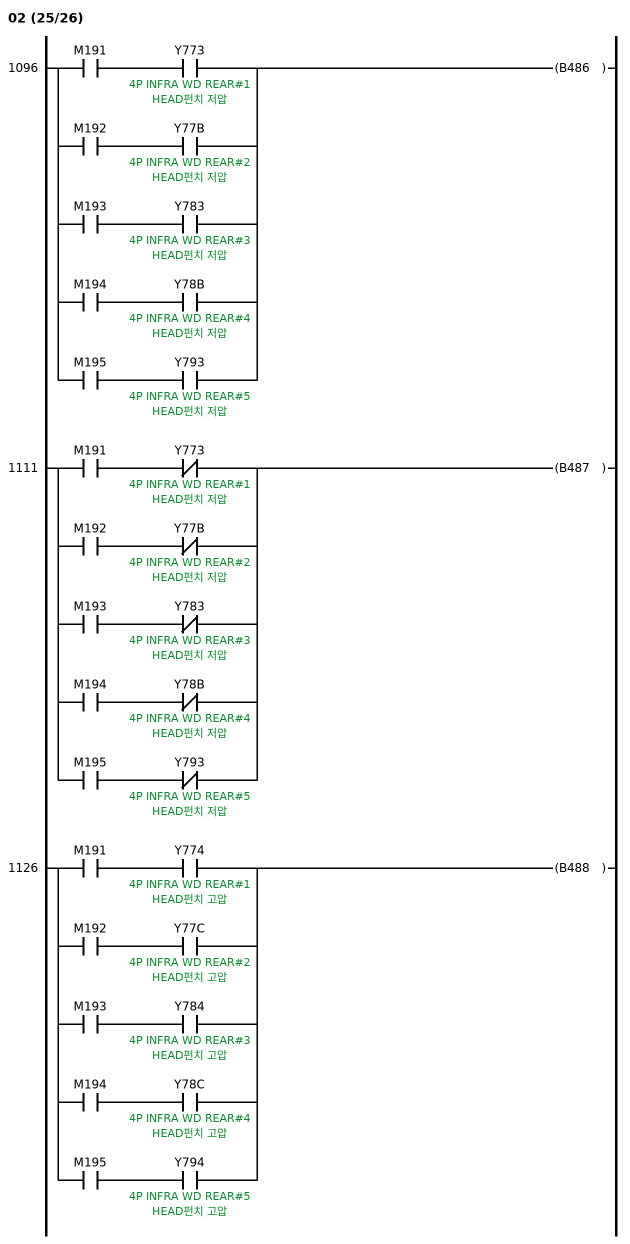
1096  LD      M191
      AND     Y773  ; 4P INFRA WD REAR#1 HEAD펀치 저압
      LD      M192
      AND     Y77B  ; 4P INFRA WD REAR#2 HEAD펀치 저압
      ORB
      LD      M193
      AND     Y783  ; 4P INFRA WD REAR#3 HEAD펀치 저압
      ORB
      LD      M194
      AND     Y78B  ; 4P INFRA WD REAR#4 HEAD펀치 저압
      ORB
      LD      M195
      AND     Y793  ; 4P INFRA WD REAR#5 HEAD펀치 저압
      ORB
      OUT     B486
1111  LD      M191
      ANI     Y773  ; 4P INFRA WD REAR#1 HEAD펀치 저압
      LD      M192
      ANI     Y77B  ; 4P INFRA WD REAR#2 HEAD펀치 저압
      ORB
      LD      M193
      ANI     Y783  ; 4P INFRA WD REAR#3 HEAD펀치 저압
      ORB
      LD      M194
      ANI     Y78B  ; 4P INFRA WD REAR#4 HEAD펀치 저압
      ORB
      LD      M195
      ANI     Y793  ; 4P INFRA WD REAR#5 HEAD펀치 저압
      ORB
      OUT     B487
1126  LD      M191
      AND     Y774  ; 4P INFRA WD REAR#1 HEAD펀치 고압
      LD      M192
      AND     Y77C  ; 4P INFRA WD REAR#2 HEAD펀치 고압
      ORB
      LD      M193
      AND     Y784  ; 4P INFRA WD REAR#3 HEAD펀치 고압
      ORB
      LD      M194
      AND     Y78C  ; 4P INFRA WD REAR#4 HEAD펀치 고압
      ORB
      LD      M195
      AND     Y794  ; 4P INFRA WD REAR#5 HEAD펀치 고압
      ORB
      OUT     B488
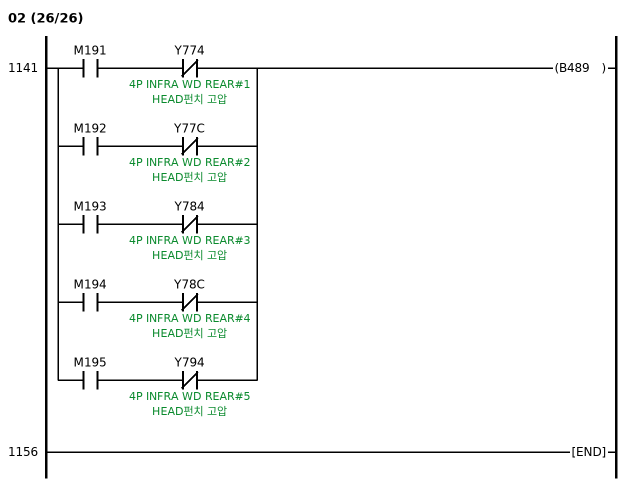
1141  LD      M191
      ANI     Y774  ; 4P INFRA WD REAR#1 HEAD펀치 고압
      LD      M192
      ANI     Y77C  ; 4P INFRA WD REAR#2 HEAD펀치 고압
      ORB
      LD      M193
      ANI     Y784  ; 4P INFRA WD REAR#3 HEAD펀치 고압
      ORB
      LD      M194
      ANI     Y78C  ; 4P INFRA WD REAR#4 HEAD펀치 고압
      ORB
      LD      M195
      ANI     Y794  ; 4P INFRA WD REAR#5 HEAD펀치 고압
      ORB
      OUT     B489
1156  END
END_PROGRAM

PROGRAM 03  // OUTPUT
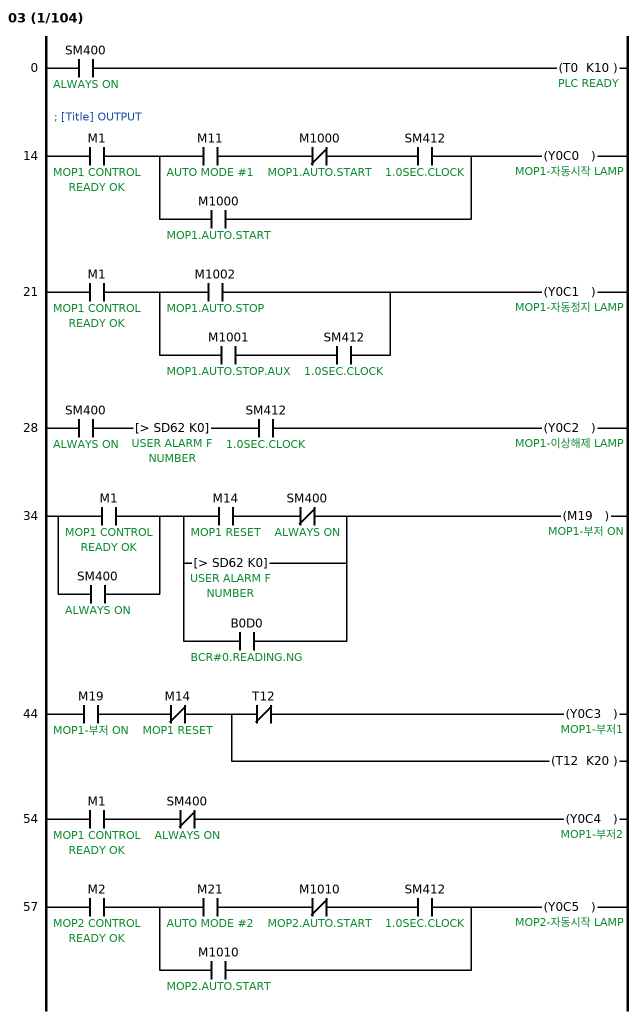
0     LD      SM400  ; ALWAYS ON
      OUT     T0 K10  ; PLC READY
; [Title] OUTPUT
14    LD      M1  ; MOP1 CONTROL READY OK
      LD      M11  ; AUTO MODE #1
      ANI     M1000  ; MOP1.AUTO.START
      AND     SM412  ; 1.0SEC.CLOCK
      OR      M1000  ; MOP1.AUTO.START
      ANB
      OUT     Y0C0  ; MOP1-자동시작 LAMP
21    LD      M1  ; MOP1 CONTROL READY OK
      LD      M1002  ; MOP1.AUTO.STOP
      LD      M1001  ; MOP1.AUTO.STOP.AUX
      AND     SM412  ; 1.0SEC.CLOCK
      ORB
      ANB
      OUT     Y0C1  ; MOP1-자동정지 LAMP
28    LD      SM400  ; ALWAYS ON
      AND>    SD62 K0  ; USER ALARM F NUMBER
      AND     SM412  ; 1.0SEC.CLOCK
      OUT     Y0C2  ; MOP1-이상해제 LAMP
34    LD      M1  ; MOP1 CONTROL READY OK
      OR      SM400  ; ALWAYS ON
      LD      M14  ; MOP1 RESET
      ANI     SM400  ; ALWAYS ON
      OR>     SD62 K0  ; USER ALARM F NUMBER
      OR      B0D0  ; BCR#0.READING.NG
      ANB
      OUT     M19  ; MOP1-부저 ON
44    LD      M19  ; MOP1-부저 ON
      ANI     M14  ; MOP1 RESET
      MPS
      ANI     T12
      OUT     Y0C3  ; MOP1-부저1
      MPP
      OUT     T12 K20
54    LD      M1  ; MOP1 CONTROL READY OK
      ANI     SM400  ; ALWAYS ON
      OUT     Y0C4  ; MOP1-부저2
57    LD      M2  ; MOP2 CONTROL READY OK
      LD      M21  ; AUTO MODE #2
      ANI     M1010  ; MOP2.AUTO.START
      AND     SM412  ; 1.0SEC.CLOCK
      OR      M1010  ; MOP2.AUTO.START
      ANB
      OUT     Y0C5  ; MOP2-자동시작 LAMP
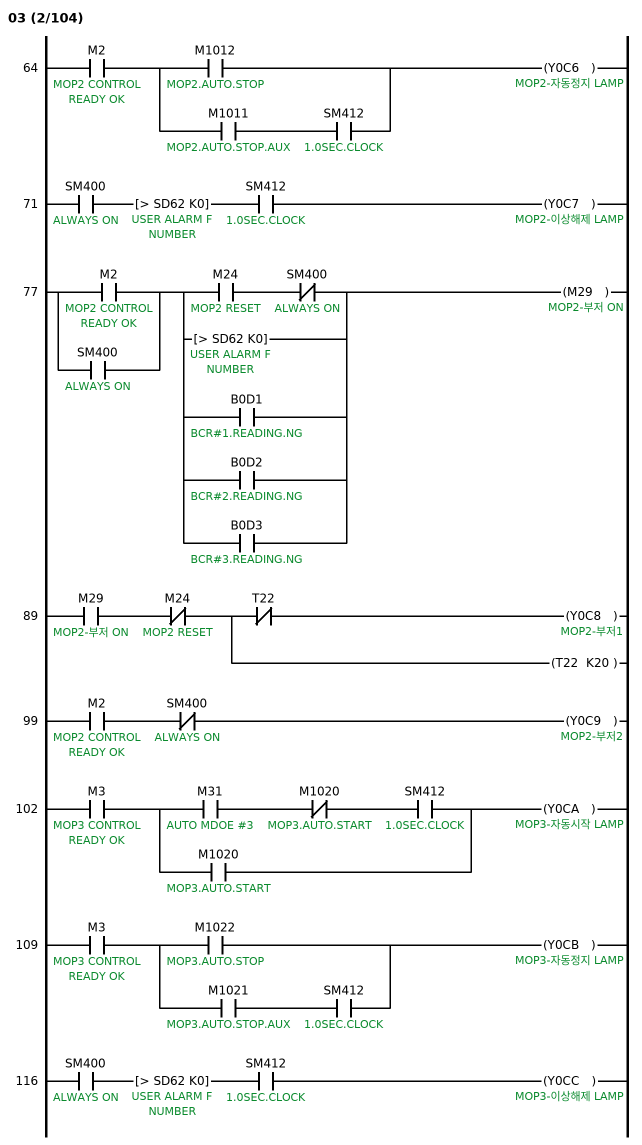
64    LD      M2  ; MOP2 CONTROL READY OK
      LD      M1012  ; MOP2.AUTO.STOP
      LD      M1011  ; MOP2.AUTO.STOP.AUX
      AND     SM412  ; 1.0SEC.CLOCK
      ORB
      ANB
      OUT     Y0C6  ; MOP2-자동정지 LAMP
71    LD      SM400  ; ALWAYS ON
      AND>    SD62 K0  ; USER ALARM F NUMBER
      AND     SM412  ; 1.0SEC.CLOCK
      OUT     Y0C7  ; MOP2-이상해제 LAMP
77    LD      M2  ; MOP2 CONTROL READY OK
      OR      SM400  ; ALWAYS ON
      LD      M24  ; MOP2 RESET
      ANI     SM400  ; ALWAYS ON
      OR>     SD62 K0  ; USER ALARM F NUMBER
      OR      B0D1  ; BCR#1.READING.NG
      OR      B0D2  ; BCR#2.READING.NG
      OR      B0D3  ; BCR#3.READING.NG
      ANB
      OUT     M29  ; MOP2-부저 ON
89    LD      M29  ; MOP2-부저 ON
      ANI     M24  ; MOP2 RESET
      MPS
      ANI     T22
      OUT     Y0C8  ; MOP2-부저1
      MPP
      OUT     T22 K20
99    LD      M2  ; MOP2 CONTROL READY OK
      ANI     SM400  ; ALWAYS ON
      OUT     Y0C9  ; MOP2-부저2
102   LD      M3  ; MOP3 CONTROL READY OK
      LD      M31  ; AUTO MDOE #3
      ANI     M1020  ; MOP3.AUTO.START
      AND     SM412  ; 1.0SEC.CLOCK
      OR      M1020  ; MOP3.AUTO.START
      ANB
      OUT     Y0CA  ; MOP3-자동시작 LAMP
109   LD      M3  ; MOP3 CONTROL READY OK
      LD      M1022  ; MOP3.AUTO.STOP
      LD      M1021  ; MOP3.AUTO.STOP.AUX
      AND     SM412  ; 1.0SEC.CLOCK
      ORB
      ANB
      OUT     Y0CB  ; MOP3-자동정지 LAMP
116   LD      SM400  ; ALWAYS ON
      AND>    SD62 K0  ; USER ALARM F NUMBER
      AND     SM412  ; 1.0SEC.CLOCK
      OUT     Y0CC  ; MOP3-이상해제 LAMP
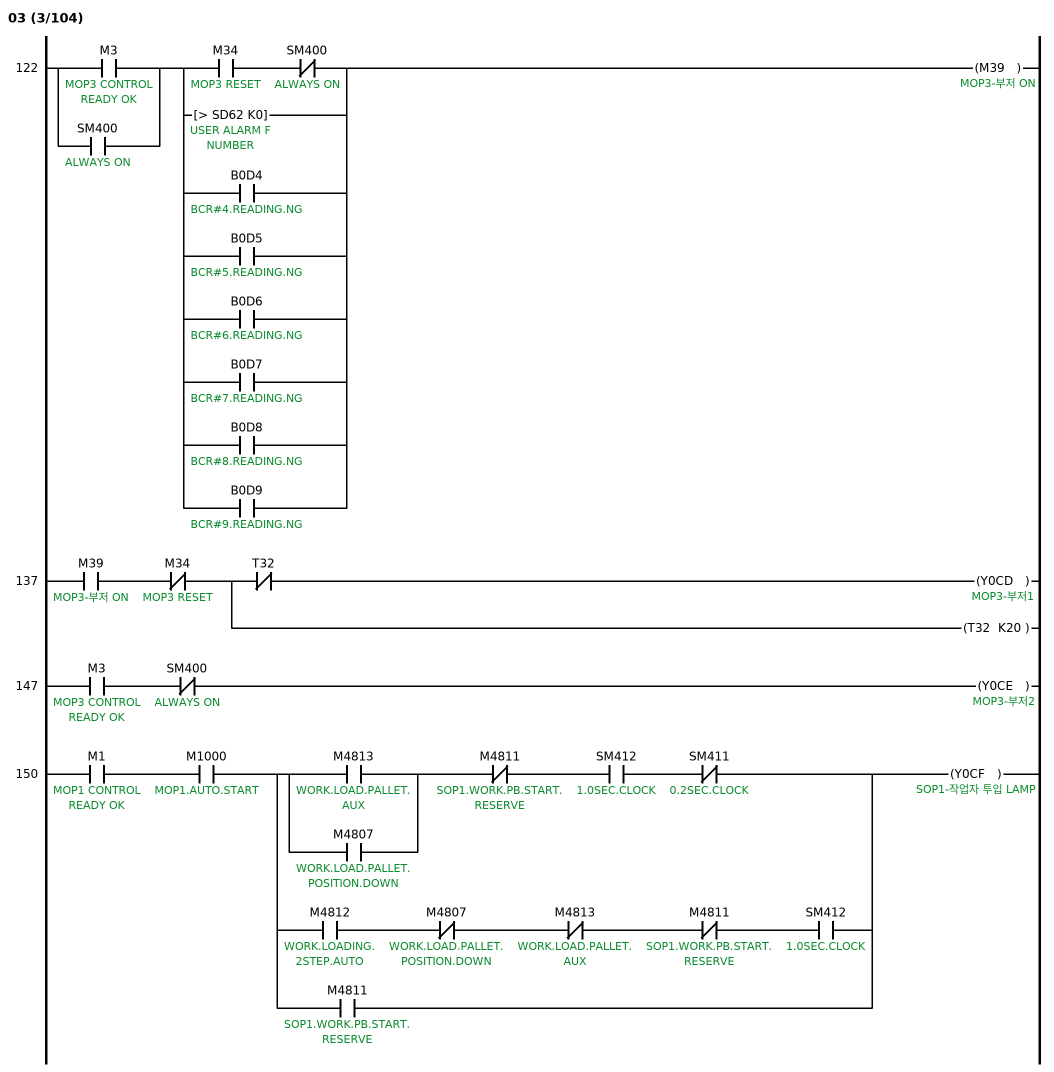
122   LD      M3  ; MOP3 CONTROL READY OK
      OR      SM400  ; ALWAYS ON
      LD      M34  ; MOP3 RESET
      ANI     SM400  ; ALWAYS ON
      OR>     SD62 K0  ; USER ALARM F NUMBER
      OR      B0D4  ; BCR#4.READING.NG
      OR      B0D5  ; BCR#5.READING.NG
      OR      B0D6  ; BCR#6.READING.NG
      OR      B0D7  ; BCR#7.READING.NG
      OR      B0D8  ; BCR#8.READING.NG
      OR      B0D9  ; BCR#9.READING.NG
      ANB
      OUT     M39  ; MOP3-부저 ON
137   LD      M39  ; MOP3-부저 ON
      ANI     M34  ; MOP3 RESET
      MPS
      ANI     T32
      OUT     Y0CD  ; MOP3-부저1
      MPP
      OUT     T32 K20
147   LD      M3  ; MOP3 CONTROL READY OK
      ANI     SM400  ; ALWAYS ON
      OUT     Y0CE  ; MOP3-부저2
150   LD      M1  ; MOP1 CONTROL READY OK
      AND     M1000  ; MOP1.AUTO.START
      LD      M4813  ; WORK.LOAD.PALLET.AUX
      OR      M4807  ; WORK.LOAD.PALLET.POSITION.DOWN
      ANI     M4811  ; SOP1.WORK.PB.START.RESERVE
      AND     SM412  ; 1.0SEC.CLOCK
      ANI     SM411  ; 0.2SEC.CLOCK
      LD      M4812  ; WORK.LOADING.2STEP.AUTO
      ANI     M4807  ; WORK.LOAD.PALLET.POSITION.DOWN
      ANI     M4813  ; WORK.LOAD.PALLET.AUX
      ANI     M4811  ; SOP1.WORK.PB.START.RESERVE
      AND     SM412  ; 1.0SEC.CLOCK
      ORB
      OR      M4811  ; SOP1.WORK.PB.START.RESERVE
      ANB
      OUT     Y0CF  ; SOP1-작업자 투입 LAMP
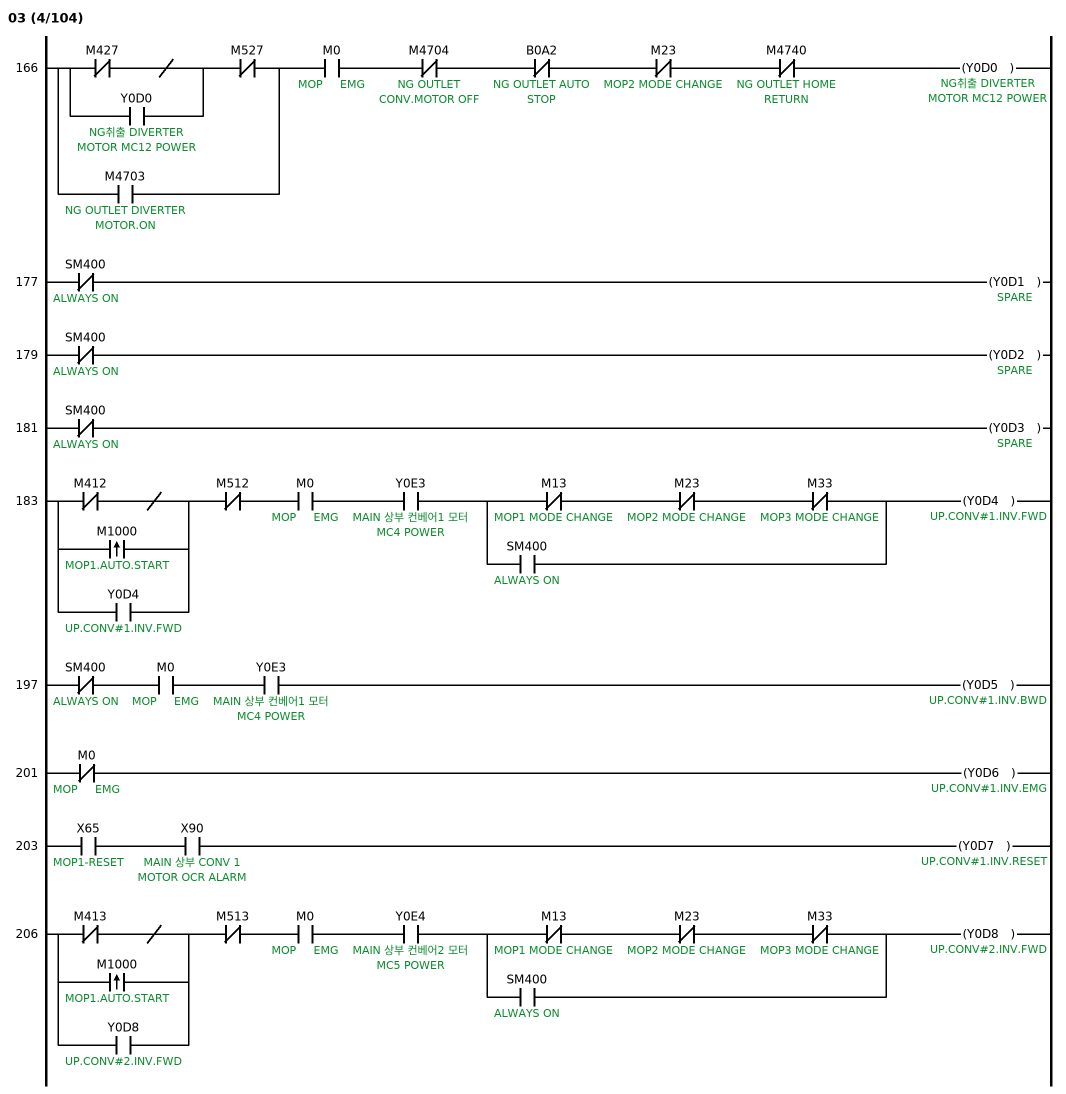
166   LDI     M427
      INV
      OR      Y0D0  ; NG취출 DIVERTER MOTOR MC12 POWER
      ANI     M527
      OR      M4703  ; NG OUTLET DIVERTER MOTOR.ON
      AND     M0  ; MOP     EMG
      ANI     M4704  ; NG OUTLET CONV.MOTOR OFF
      ANI     B0A2  ; NG OUTLET AUTO STOP
      ANI     M23  ; MOP2 MODE CHANGE
      ANI     M4740  ; NG OUTLET HOME RETURN
      OUT     Y0D0  ; NG취출 DIVERTER MOTOR MC12 POWER
177   LDI     SM400  ; ALWAYS ON
      OUT     Y0D1  ; SPARE
179   LDI     SM400  ; ALWAYS ON
      OUT     Y0D2  ; SPARE
181   LDI     SM400  ; ALWAYS ON
      OUT     Y0D3  ; SPARE
183   LDI     M412
      INV
      ORP     M1000  ; MOP1.AUTO.START
      OR      Y0D4  ; UP.CONV#1.INV.FWD
      ANI     M512
      AND     M0  ; MOP     EMG
      AND     Y0E3  ; MAIN 상부 컨베어1 모터 MC4 POWER
      LDI     M13  ; MOP1 MODE CHANGE
      ANI     M23  ; MOP2 MODE CHANGE
      ANI     M33  ; MOP3 MODE CHANGE
      OR      SM400  ; ALWAYS ON
      ANB
      OUT     Y0D4  ; UP.CONV#1.INV.FWD
197   LDI     SM400  ; ALWAYS ON
      AND     M0  ; MOP     EMG
      AND     Y0E3  ; MAIN 상부 컨베어1 모터 MC4 POWER
      OUT     Y0D5  ; UP.CONV#1.INV.BWD
201   LDI     M0  ; MOP     EMG
      OUT     Y0D6  ; UP.CONV#1.INV.EMG
203   LD      X65  ; MOP1-RESET
      AND     X90  ; MAIN 상부 CONV 1 MOTOR OCR ALARM
      OUT     Y0D7  ; UP.CONV#1.INV.RESET
206   LDI     M413
      INV
      ORP     M1000  ; MOP1.AUTO.START
      OR      Y0D8  ; UP.CONV#2.INV.FWD
      ANI     M513
      AND     M0  ; MOP     EMG
      AND     Y0E4  ; MAIN 상부 컨베어2 모터 MC5 POWER
      LDI     M13  ; MOP1 MODE CHANGE
      ANI     M23  ; MOP2 MODE CHANGE
      ANI     M33  ; MOP3 MODE CHANGE
      OR      SM400  ; ALWAYS ON
      ANB
      OUT     Y0D8  ; UP.CONV#2.INV.FWD
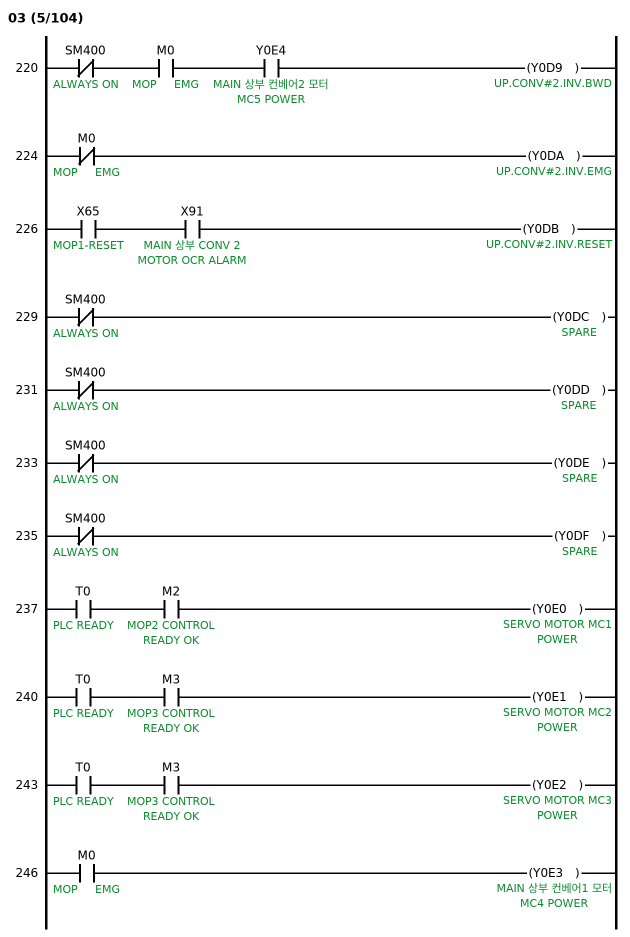
220   LDI     SM400  ; ALWAYS ON
      AND     M0  ; MOP     EMG
      AND     Y0E4  ; MAIN 상부 컨베어2 모터 MC5 POWER
      OUT     Y0D9  ; UP.CONV#2.INV.BWD
224   LDI     M0  ; MOP     EMG
      OUT     Y0DA  ; UP.CONV#2.INV.EMG
226   LD      X65  ; MOP1-RESET
      AND     X91  ; MAIN 상부 CONV 2 MOTOR OCR ALARM
      OUT     Y0DB  ; UP.CONV#2.INV.RESET
229   LDI     SM400  ; ALWAYS ON
      OUT     Y0DC  ; SPARE
231   LDI     SM400  ; ALWAYS ON
      OUT     Y0DD  ; SPARE
233   LDI     SM400  ; ALWAYS ON
      OUT     Y0DE  ; SPARE
235   LDI     SM400  ; ALWAYS ON
      OUT     Y0DF  ; SPARE
237   LD      T0  ; PLC READY
      AND     M2  ; MOP2 CONTROL READY OK
      OUT     Y0E0  ; SERVO MOTOR MC1 POWER
240   LD      T0  ; PLC READY
      AND     M3  ; MOP3 CONTROL READY OK
      OUT     Y0E1  ; SERVO MOTOR MC2 POWER
243   LD      T0  ; PLC READY
      AND     M3  ; MOP3 CONTROL READY OK
      OUT     Y0E2  ; SERVO MOTOR MC3 POWER
246   LD      M0  ; MOP     EMG
      OUT     Y0E3  ; MAIN 상부 컨베어1 모터 MC4 POWER
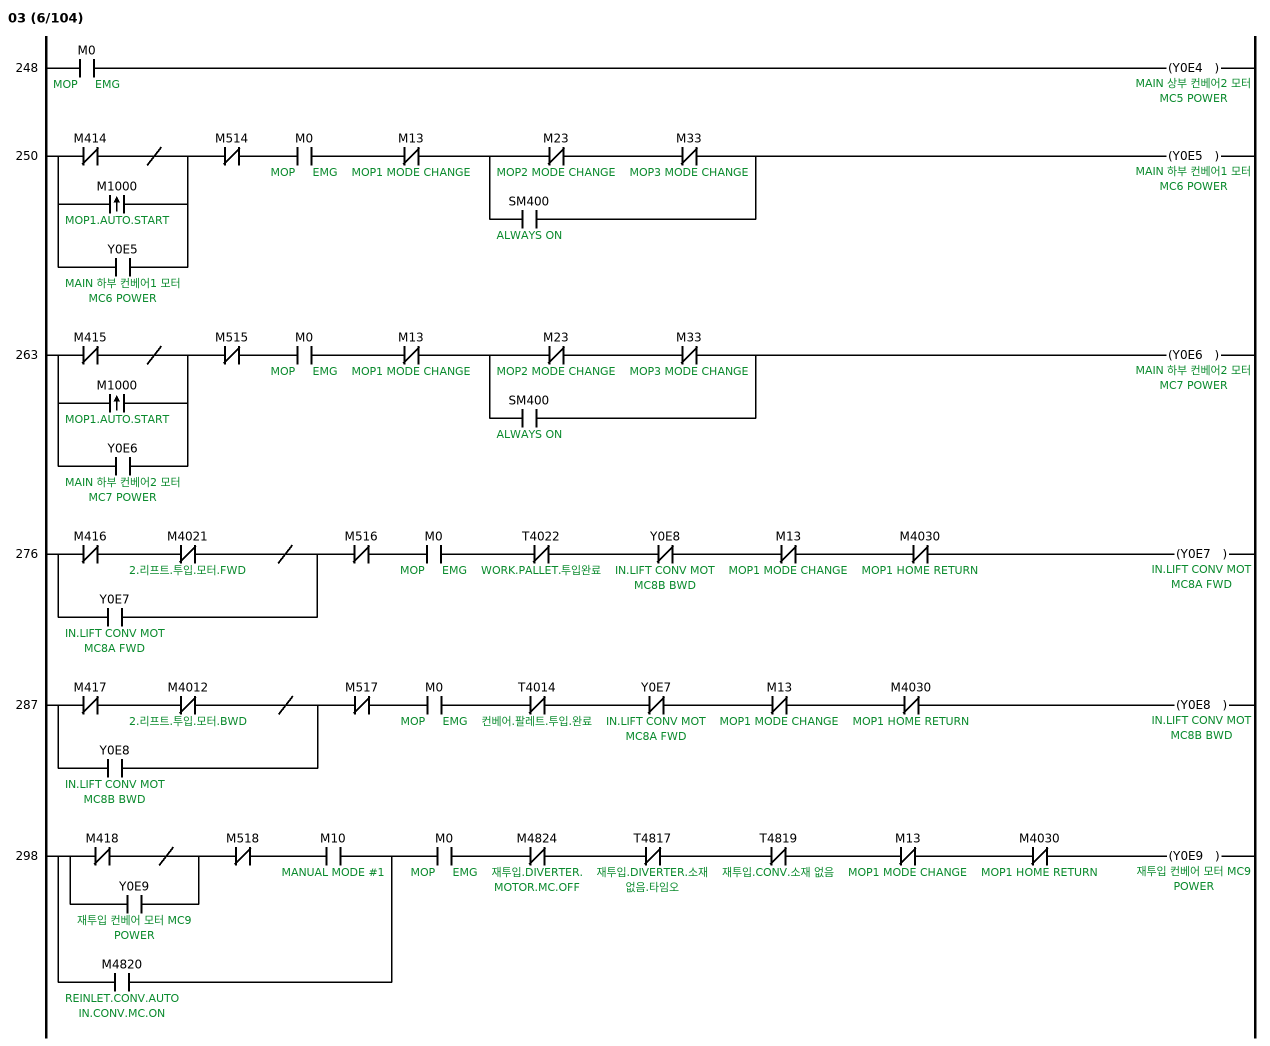
248   LD      M0  ; MOP     EMG
      OUT     Y0E4  ; MAIN 상부 컨베어2 모터 MC5 POWER
250   LDI     M414
      INV
      ORP     M1000  ; MOP1.AUTO.START
      OR      Y0E5  ; MAIN 하부 컨베어1 모터 MC6 POWER
      ANI     M514
      AND     M0  ; MOP     EMG
      ANI     M13  ; MOP1 MODE CHANGE
      LDI     M23  ; MOP2 MODE CHANGE
      ANI     M33  ; MOP3 MODE CHANGE
      OR      SM400  ; ALWAYS ON
      ANB
      OUT     Y0E5  ; MAIN 하부 컨베어1 모터 MC6 POWER
263   LDI     M415
      INV
      ORP     M1000  ; MOP1.AUTO.START
      OR      Y0E6  ; MAIN 하부 컨베어2 모터 MC7 POWER
      ANI     M515
      AND     M0  ; MOP     EMG
      ANI     M13  ; MOP1 MODE CHANGE
      LDI     M23  ; MOP2 MODE CHANGE
      ANI     M33  ; MOP3 MODE CHANGE
      OR      SM400  ; ALWAYS ON
      ANB
      OUT     Y0E6  ; MAIN 하부 컨베어2 모터 MC7 POWER
276   LDI     M416
      ANI     M4021  ; 2.리프트.투입.모터.FWD
      INV
      OR      Y0E7  ; IN.LIFT CONV MOT MC8A FWD
      ANI     M516
      AND     M0  ; MOP     EMG
      ANI     T4022  ; WORK.PALLET.투입완료
      ANI     Y0E8  ; IN.LIFT CONV MOT MC8B BWD
      ANI     M13  ; MOP1 MODE CHANGE
      ANI     M4030  ; MOP1 HOME RETURN
      OUT     Y0E7  ; IN.LIFT CONV MOT MC8A FWD
287   LDI     M417
      ANI     M4012  ; 2.리프트.투입.모터.BWD
      INV
      OR      Y0E8  ; IN.LIFT CONV MOT MC8B BWD
      ANI     M517
      AND     M0  ; MOP     EMG
      ANI     T4014  ; 컨베어.팔레트.투입.완료
      ANI     Y0E7  ; IN.LIFT CONV MOT MC8A FWD
      ANI     M13  ; MOP1 MODE CHANGE
      ANI     M4030  ; MOP1 HOME RETURN
      OUT     Y0E8  ; IN.LIFT CONV MOT MC8B BWD
298   LDI     M418
      INV
      OR      Y0E9  ; 재투입 컨베어 모터 MC9 POWER
      ANI     M518
      AND     M10  ; MANUAL MODE #1
      OR      M4820  ; REINLET.CONV.AUTO IN.CONV.MC.ON
      AND     M0  ; MOP     EMG
      ANI     M4824  ; 재투입.DIVERTER.MOTOR.MC.OFF
      ANI     T4817  ; 재투입.DIVERTER.소재 없음.타임오
      ANI     T4819  ; 재투입.CONV.소재 없음
      ANI     M13  ; MOP1 MODE CHANGE
      ANI     M4030  ; MOP1 HOME RETURN
      OUT     Y0E9  ; 재투입 컨베어 모터 MC9 POWER
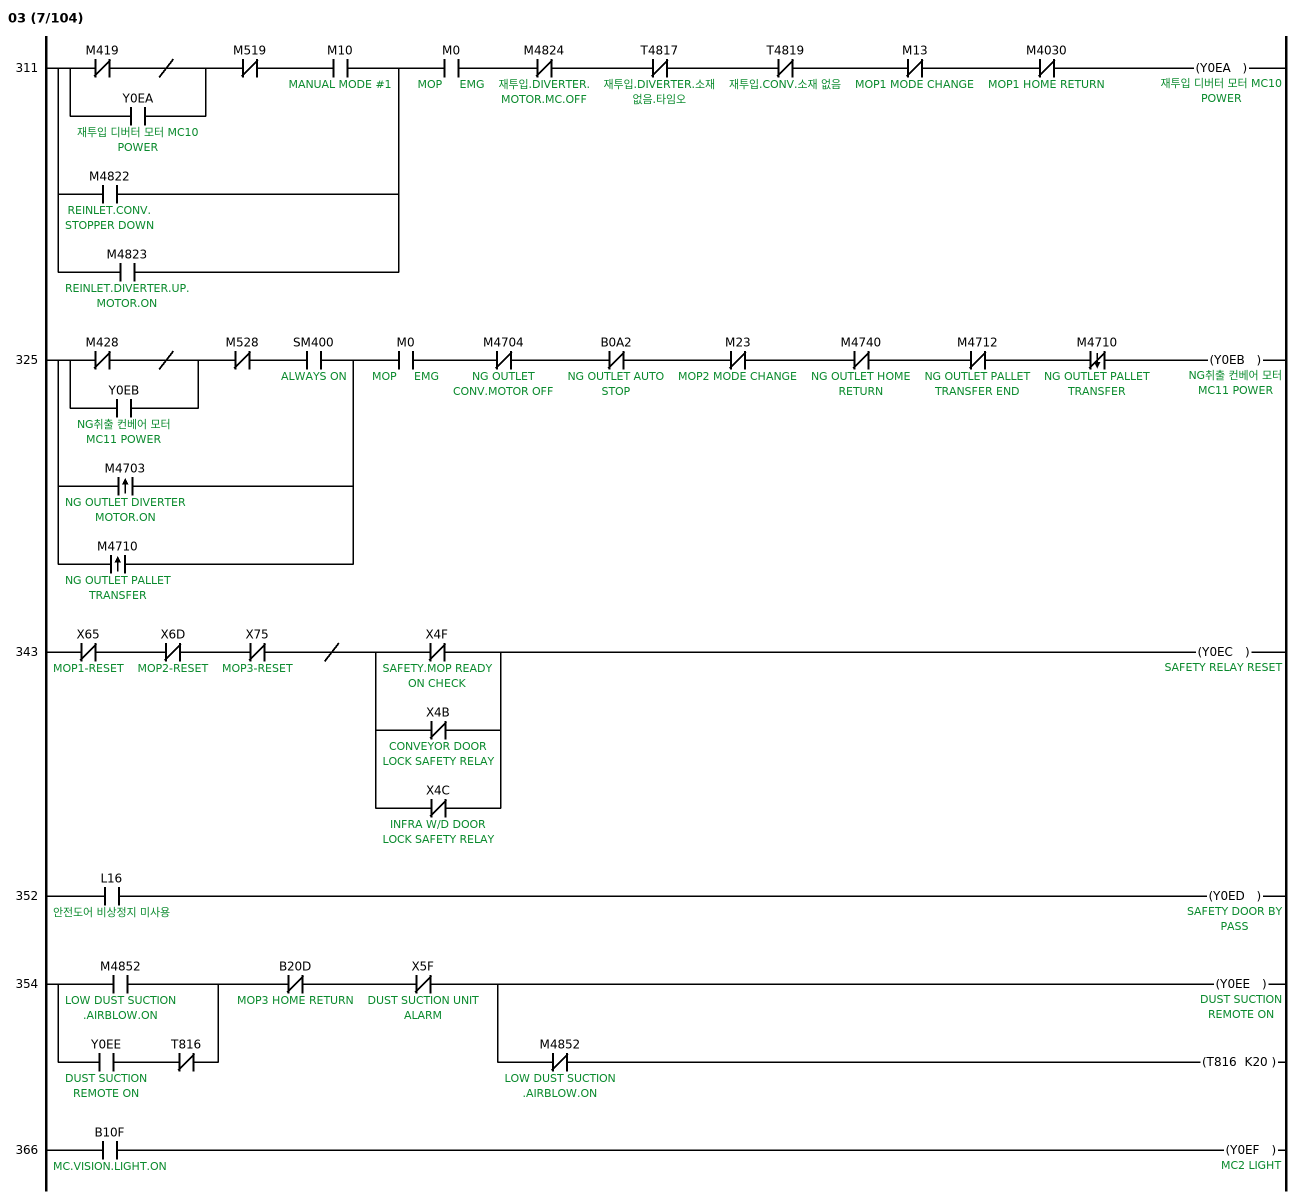
311   LDI     M419
      INV
      OR      Y0EA  ; 재투입 디버터 모터 MC10 POWER
      ANI     M519
      AND     M10  ; MANUAL MODE #1
      OR      M4822  ; REINLET.CONV.STOPPER DOWN
      OR      M4823  ; REINLET.DIVERTER.UP.MOTOR.ON
      AND     M0  ; MOP     EMG
      ANI     M4824  ; 재투입.DIVERTER.MOTOR.MC.OFF
      ANI     T4817  ; 재투입.DIVERTER.소재 없음.타임오
      ANI     T4819  ; 재투입.CONV.소재 없음
      ANI     M13  ; MOP1 MODE CHANGE
      ANI     M4030  ; MOP1 HOME RETURN
      OUT     Y0EA  ; 재투입 디버터 모터 MC10 POWER
325   LDI     M428
      INV
      OR      Y0EB  ; NG취출 컨베어 모터 MC11 POWER
      ANI     M528
      AND     SM400  ; ALWAYS ON
      ORP     M4703  ; NG OUTLET DIVERTER MOTOR.ON
      ORP     M4710  ; NG OUTLET PALLET TRANSFER
      AND     M0  ; MOP     EMG
      ANI     M4704  ; NG OUTLET CONV.MOTOR OFF
      ANI     B0A2  ; NG OUTLET AUTO STOP
      ANI     M23  ; MOP2 MODE CHANGE
      ANI     M4740  ; NG OUTLET HOME RETURN
      ANI     M4712  ; NG OUTLET PALLET TRANSFER END
      ANDFI   M4710  ; NG OUTLET PALLET TRANSFER
      OUT     Y0EB  ; NG취출 컨베어 모터 MC11 POWER
343   LDI     X65  ; MOP1-RESET
      ANI     X6D  ; MOP2-RESET
      ANI     X75  ; MOP3-RESET
      INV
      LDI     X4F  ; SAFETY.MOP READY ON CHECK
      ORI     X4B  ; CONVEYOR DOOR LOCK SAFETY RELAY
      ORI     X4C  ; INFRA W/D DOOR LOCK SAFETY RELAY
      ANB
      OUT     Y0EC  ; SAFETY RELAY RESET
352   LD      L16  ; 안전도어 비상정지 미사용
      OUT     Y0ED  ; SAFETY DOOR BY PASS
354   LD      M4852  ; LOW DUST SUCTION .AIRBLOW.ON
      LD      Y0EE  ; DUST SUCTION REMOTE ON
      ANI     T816
      ORB
      ANI     B20D  ; MOP3 HOME RETURN
      ANI     X5F  ; DUST SUCTION UNIT ALARM
      OUT     Y0EE  ; DUST SUCTION REMOTE ON
      ANI     M4852  ; LOW DUST SUCTION .AIRBLOW.ON
      OUT     T816 K20
366   LD      B10F  ; MC.VISION.LIGHT.ON
      OUT     Y0EF  ; MC2 LIGHT
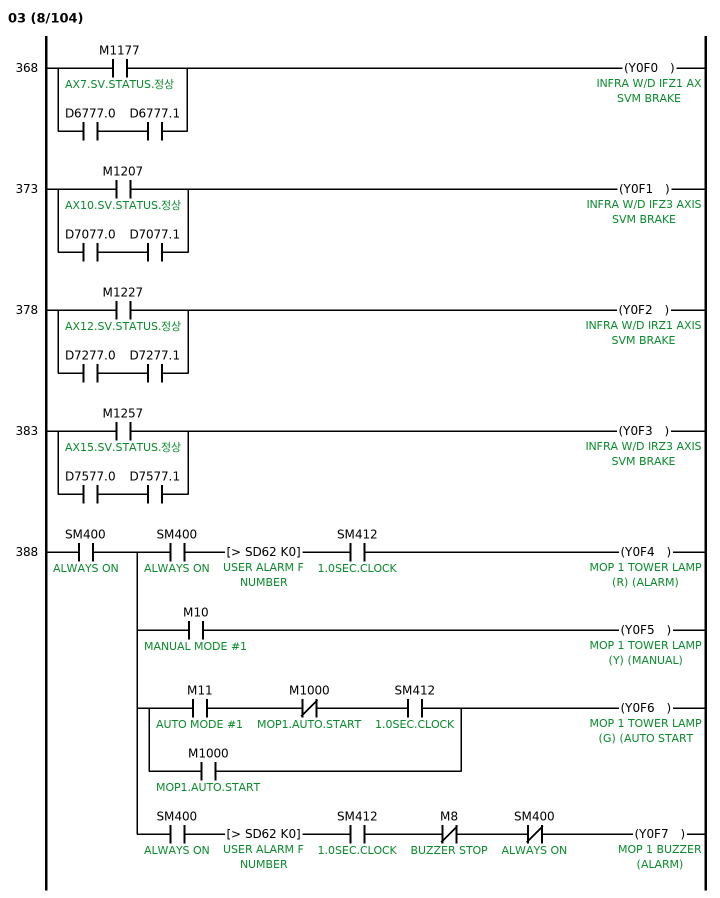
368   LD      M1177  ; AX7.SV.STATUS.정상
      LD      D6777.0
      AND     D6777.1
      ORB
      OUT     Y0F0  ; INFRA W/D IFZ1 AX SVM BRAKE
373   LD      M1207  ; AX10.SV.STATUS.정상
      LD      D7077.0
      AND     D7077.1
      ORB
      OUT     Y0F1  ; INFRA W/D IFZ3 AXIS SVM BRAKE
378   LD      M1227  ; AX12.SV.STATUS.정상
      LD      D7277.0
      AND     D7277.1
      ORB
      OUT     Y0F2  ; INFRA W/D IRZ1 AXIS SVM BRAKE
383   LD      M1257  ; AX15.SV.STATUS.정상
      LD      D7577.0
      AND     D7577.1
      ORB
      OUT     Y0F3  ; INFRA W/D IRZ3 AXIS SVM BRAKE
388   LD      SM400  ; ALWAYS ON
      MPS
      AND     SM400  ; ALWAYS ON
      AND>    SD62 K0  ; USER ALARM F NUMBER
      AND     SM412  ; 1.0SEC.CLOCK
      OUT     Y0F4  ; MOP 1 TOWER LAMP (R) (ALARM)
      MRD
      AND     M10  ; MANUAL MODE #1
      OUT     Y0F5  ; MOP 1 TOWER LAMP (Y) (MANUAL)
      MRD
      LD      M11  ; AUTO MODE #1
      ANI     M1000  ; MOP1.AUTO.START
      AND     SM412  ; 1.0SEC.CLOCK
      OR      M1000  ; MOP1.AUTO.START
      ANB
      OUT     Y0F6  ; MOP 1 TOWER LAMP (G) (AUTO START
      MPP
      AND     SM400  ; ALWAYS ON
      AND>    SD62 K0  ; USER ALARM F NUMBER
      AND     SM412  ; 1.0SEC.CLOCK
      ANI     M8  ; BUZZER STOP
      ANI     SM400  ; ALWAYS ON
      OUT     Y0F7  ; MOP 1 BUZZER (ALARM)
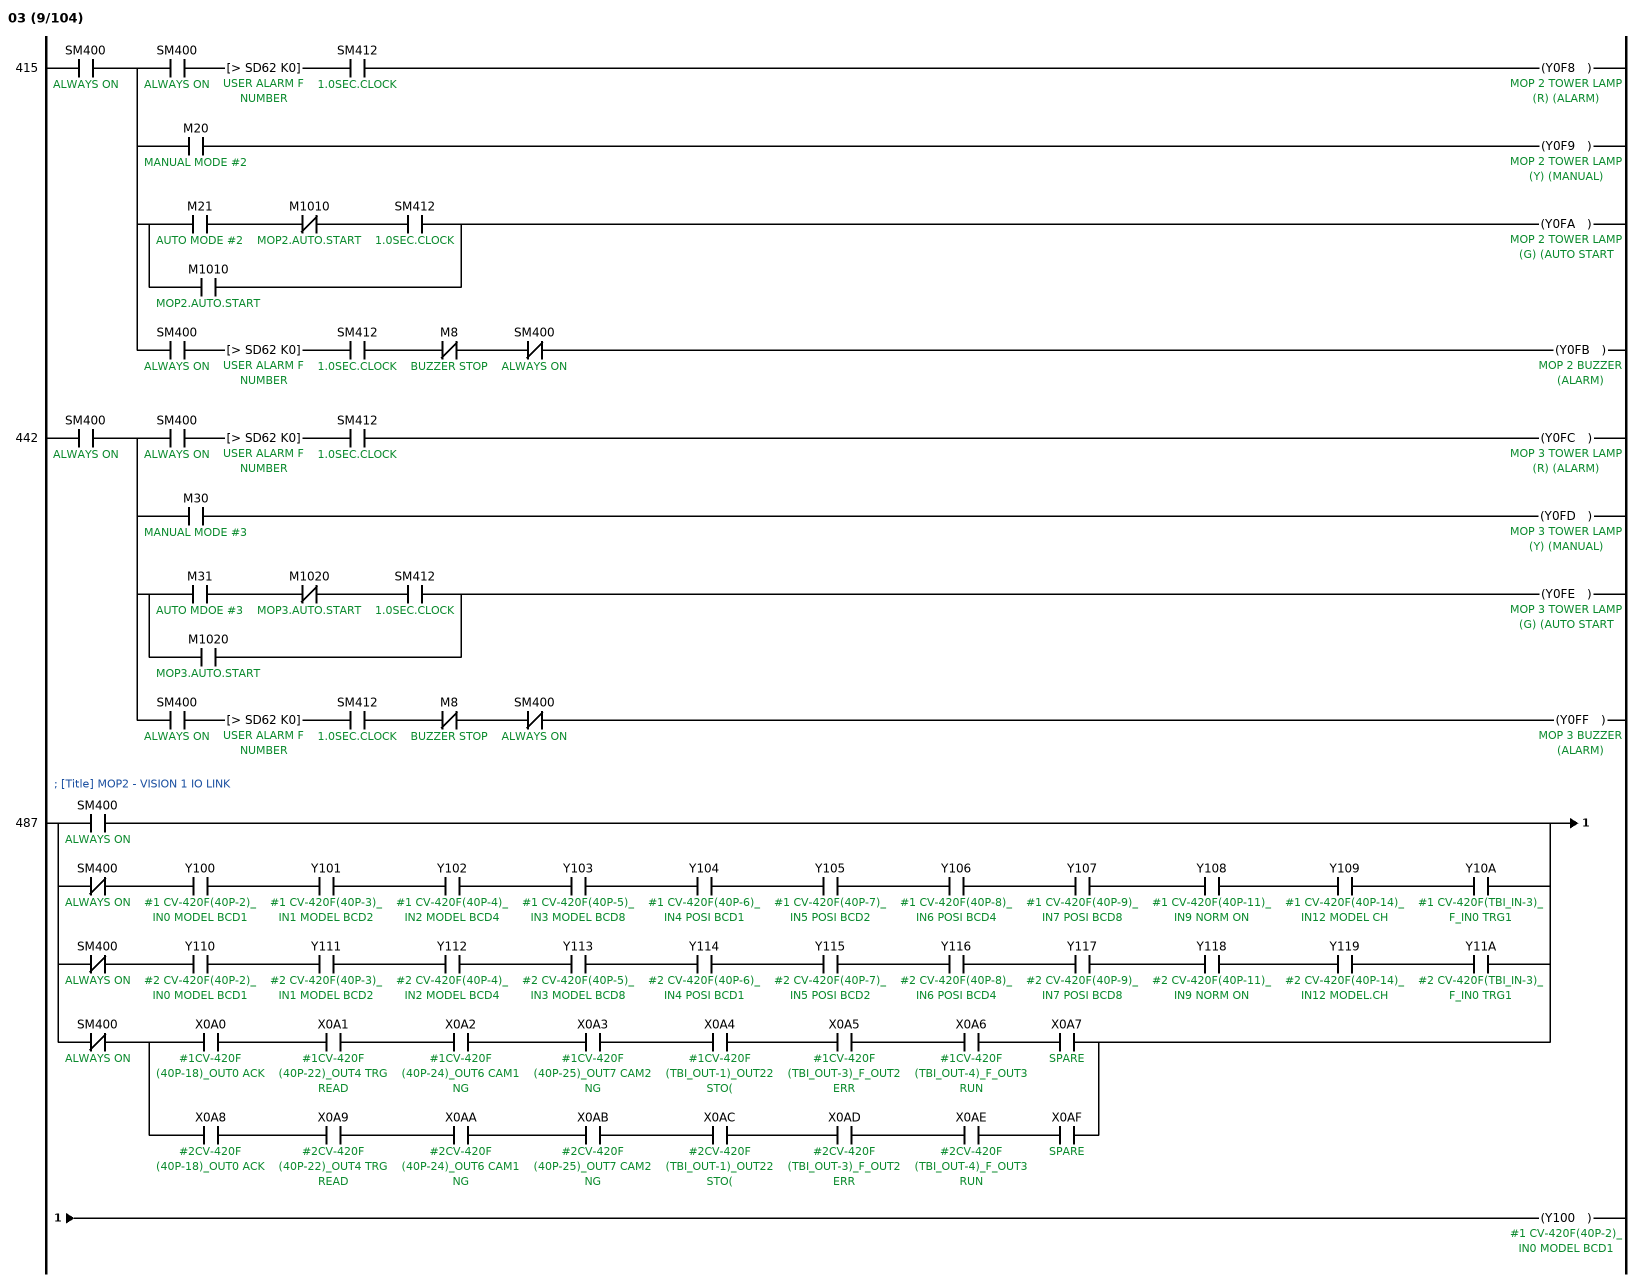
415   LD      SM400  ; ALWAYS ON
      MPS
      AND     SM400  ; ALWAYS ON
      AND>    SD62 K0  ; USER ALARM F NUMBER
      AND     SM412  ; 1.0SEC.CLOCK
      OUT     Y0F8  ; MOP 2 TOWER LAMP (R) (ALARM)
      MRD
      AND     M20  ; MANUAL MODE #2
      OUT     Y0F9  ; MOP 2 TOWER LAMP (Y) (MANUAL)
      MRD
      LD      M21  ; AUTO MODE #2
      ANI     M1010  ; MOP2.AUTO.START
      AND     SM412  ; 1.0SEC.CLOCK
      OR      M1010  ; MOP2.AUTO.START
      ANB
      OUT     Y0FA  ; MOP 2 TOWER LAMP (G) (AUTO START
      MPP
      AND     SM400  ; ALWAYS ON
      AND>    SD62 K0  ; USER ALARM F NUMBER
      AND     SM412  ; 1.0SEC.CLOCK
      ANI     M8  ; BUZZER STOP
      ANI     SM400  ; ALWAYS ON
      OUT     Y0FB  ; MOP 2 BUZZER (ALARM)
442   LD      SM400  ; ALWAYS ON
      MPS
      AND     SM400  ; ALWAYS ON
      AND>    SD62 K0  ; USER ALARM F NUMBER
      AND     SM412  ; 1.0SEC.CLOCK
      OUT     Y0FC  ; MOP 3 TOWER LAMP (R) (ALARM)
      MRD
      AND     M30  ; MANUAL MODE #3
      OUT     Y0FD  ; MOP 3 TOWER LAMP (Y) (MANUAL)
      MRD
      LD      M31  ; AUTO MDOE #3
      ANI     M1020  ; MOP3.AUTO.START
      AND     SM412  ; 1.0SEC.CLOCK
      OR      M1020  ; MOP3.AUTO.START
      ANB
      OUT     Y0FE  ; MOP 3 TOWER LAMP (G) (AUTO START
      MPP
      AND     SM400  ; ALWAYS ON
      AND>    SD62 K0  ; USER ALARM F NUMBER
      AND     SM412  ; 1.0SEC.CLOCK
      ANI     M8  ; BUZZER STOP
      ANI     SM400  ; ALWAYS ON
      OUT     Y0FF  ; MOP 3 BUZZER (ALARM)
; [Title] MOP2 - VISION 1 IO LINK
487   LD      SM400  ; ALWAYS ON
      LDI     SM400  ; ALWAYS ON
      AND     Y100  ; #1 CV-420F(40P-2)_IN0 MODEL BCD1
      AND     Y101  ; #1 CV-420F(40P-3)_IN1 MODEL BCD2
      AND     Y102  ; #1 CV-420F(40P-4)_IN2 MODEL BCD4
      AND     Y103  ; #1 CV-420F(40P-5)_IN3 MODEL BCD8
      AND     Y104  ; #1 CV-420F(40P-6)_IN4 POSI BCD1
      AND     Y105  ; #1 CV-420F(40P-7)_IN5 POSI BCD2
      AND     Y106  ; #1 CV-420F(40P-8)_IN6 POSI BCD4
      AND     Y107  ; #1 CV-420F(40P-9)_IN7 POSI BCD8
      AND     Y108  ; #1 CV-420F(40P-11)_IN9 NORM ON
      AND     Y109  ; #1 CV-420F(40P-14)_IN12 MODEL CH
      AND     Y10A  ; #1 CV-420F(TBI_IN-3)_F_IN0 TRG1
      ORB
      LDI     SM400  ; ALWAYS ON
      AND     Y110  ; #2 CV-420F(40P-2)_IN0 MODEL BCD1
      AND     Y111  ; #2 CV-420F(40P-3)_IN1 MODEL BCD2
      AND     Y112  ; #2 CV-420F(40P-4)_IN2 MODEL BCD4
      AND     Y113  ; #2 CV-420F(40P-5)_IN3 MODEL BCD8
      AND     Y114  ; #2 CV-420F(40P-6)_IN4 POSI BCD1
      AND     Y115  ; #2 CV-420F(40P-7)_IN5 POSI BCD2
      AND     Y116  ; #2 CV-420F(40P-8)_IN6 POSI BCD4
      AND     Y117  ; #2 CV-420F(40P-9)_IN7 POSI BCD8
      AND     Y118  ; #2 CV-420F(40P-11)_IN9 NORM ON
      AND     Y119  ; #2 CV-420F(40P-14)_IN12 MODEL.CH
      AND     Y11A  ; #2 CV-420F(TBI_IN-3)_F_IN0 TRG1
      ORB
      LDI     SM400  ; ALWAYS ON
      LD      X0A0  ; #1CV-420F (40P-18)_OUT0 ACK
      AND     X0A1  ; #1CV-420F (40P-22)_OUT4 TRG READ
      AND     X0A2  ; #1CV-420F (40P-24)_OUT6 CAM1 NG
      AND     X0A3  ; #1CV-420F (40P-25)_OUT7 CAM2 NG
      AND     X0A4  ; #1CV-420F (TBI_OUT-1)_OUT22 STO(
      AND     X0A5  ; #1CV-420F (TBI_OUT-3)_F_OUT2 ERR
      AND     X0A6  ; #1CV-420F (TBI_OUT-4)_F_OUT3 RUN
      AND     X0A7  ; SPARE
      LD      X0A8  ; #2CV-420F (40P-18)_OUT0 ACK
      AND     X0A9  ; #2CV-420F (40P-22)_OUT4 TRG READ
      AND     X0AA  ; #2CV-420F (40P-24)_OUT6 CAM1 NG
      AND     X0AB  ; #2CV-420F (40P-25)_OUT7 CAM2 NG
      AND     X0AC  ; #2CV-420F (TBI_OUT-1)_OUT22 STO(
      AND     X0AD  ; #2CV-420F (TBI_OUT-3)_F_OUT2 ERR
      AND     X0AE  ; #2CV-420F (TBI_OUT-4)_F_OUT3 RUN
      AND     X0AF  ; SPARE
      ORB
      ANB
      ORB
      OUT     Y100  ; #1 CV-420F(40P-2)_IN0 MODEL BCD1
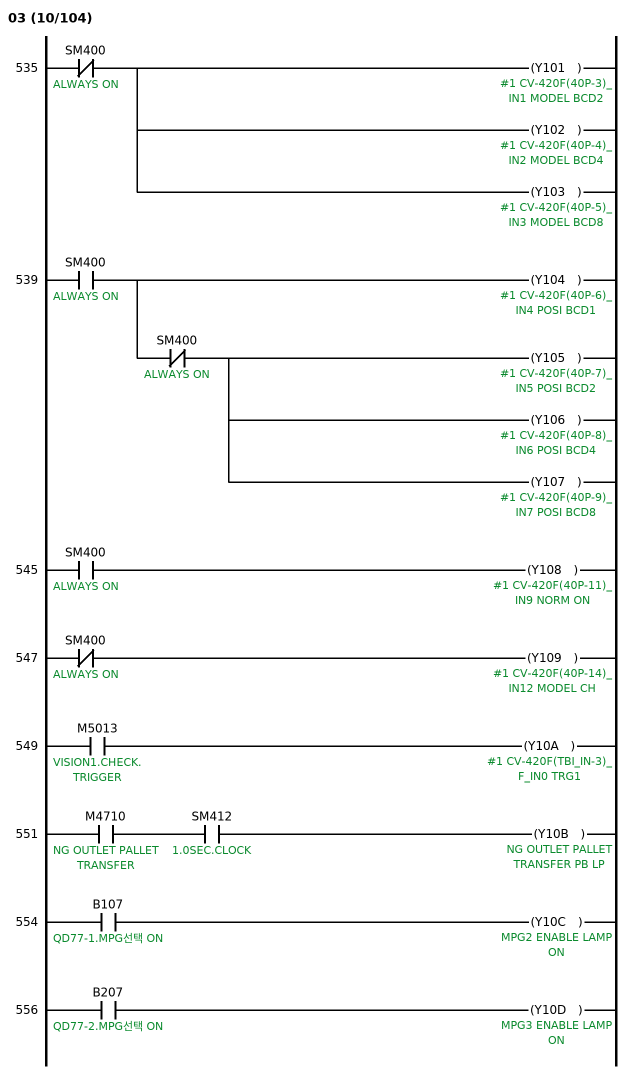
535   LDI     SM400  ; ALWAYS ON
      OUT     Y101  ; #1 CV-420F(40P-3)_IN1 MODEL BCD2
      OUT     Y102  ; #1 CV-420F(40P-4)_IN2 MODEL BCD4
      OUT     Y103  ; #1 CV-420F(40P-5)_IN3 MODEL BCD8
539   LD      SM400  ; ALWAYS ON
      OUT     Y104  ; #1 CV-420F(40P-6)_IN4 POSI BCD1
      ANI     SM400  ; ALWAYS ON
      OUT     Y105  ; #1 CV-420F(40P-7)_IN5 POSI BCD2
      OUT     Y106  ; #1 CV-420F(40P-8)_IN6 POSI BCD4
      OUT     Y107  ; #1 CV-420F(40P-9)_IN7 POSI BCD8
545   LD      SM400  ; ALWAYS ON
      OUT     Y108  ; #1 CV-420F(40P-11)_IN9 NORM ON
547   LDI     SM400  ; ALWAYS ON
      OUT     Y109  ; #1 CV-420F(40P-14)_IN12 MODEL CH
549   LD      M5013  ; VISION1.CHECK.TRIGGER
      OUT     Y10A  ; #1 CV-420F(TBI_IN-3)_F_IN0 TRG1
551   LD      M4710  ; NG OUTLET PALLET TRANSFER
      AND     SM412  ; 1.0SEC.CLOCK
      OUT     Y10B  ; NG OUTLET PALLET TRANSFER PB LP
554   LD      B107  ; QD77-1.MPG선택 ON
      OUT     Y10C  ; MPG2 ENABLE LAMP ON
556   LD      B207  ; QD77-2.MPG선택 ON
      OUT     Y10D  ; MPG3 ENABLE LAMP ON
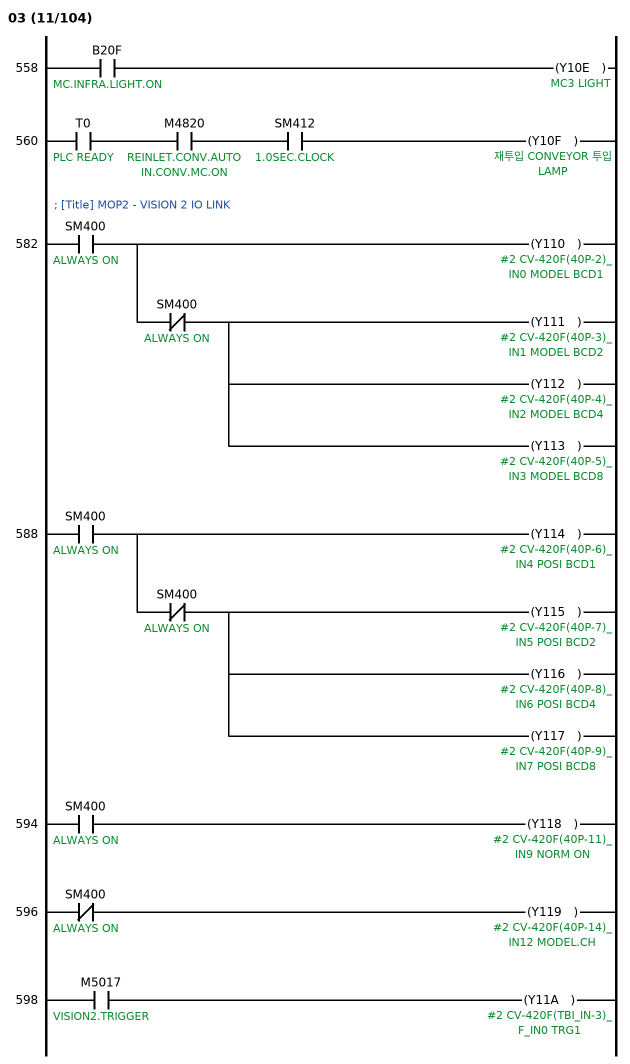
558   LD      B20F  ; MC.INFRA.LIGHT.ON
      OUT     Y10E  ; MC3 LIGHT
560   LD      T0  ; PLC READY
      AND     M4820  ; REINLET.CONV.AUTO IN.CONV.MC.ON
      AND     SM412  ; 1.0SEC.CLOCK
      OUT     Y10F  ; 재투입 CONVEYOR 투입 LAMP
; [Title] MOP2 - VISION 2 IO LINK
582   LD      SM400  ; ALWAYS ON
      OUT     Y110  ; #2 CV-420F(40P-2)_IN0 MODEL BCD1
      ANI     SM400  ; ALWAYS ON
      OUT     Y111  ; #2 CV-420F(40P-3)_IN1 MODEL BCD2
      OUT     Y112  ; #2 CV-420F(40P-4)_IN2 MODEL BCD4
      OUT     Y113  ; #2 CV-420F(40P-5)_IN3 MODEL BCD8
588   LD      SM400  ; ALWAYS ON
      OUT     Y114  ; #2 CV-420F(40P-6)_IN4 POSI BCD1
      ANI     SM400  ; ALWAYS ON
      OUT     Y115  ; #2 CV-420F(40P-7)_IN5 POSI BCD2
      OUT     Y116  ; #2 CV-420F(40P-8)_IN6 POSI BCD4
      OUT     Y117  ; #2 CV-420F(40P-9)_IN7 POSI BCD8
594   LD      SM400  ; ALWAYS ON
      OUT     Y118  ; #2 CV-420F(40P-11)_IN9 NORM ON
596   LDI     SM400  ; ALWAYS ON
      OUT     Y119  ; #2 CV-420F(40P-14)_IN12 MODEL.CH
598   LD      M5017  ; VISION2.TRIGGER
      OUT     Y11A  ; #2 CV-420F(TBI_IN-3)_F_IN0 TRG1
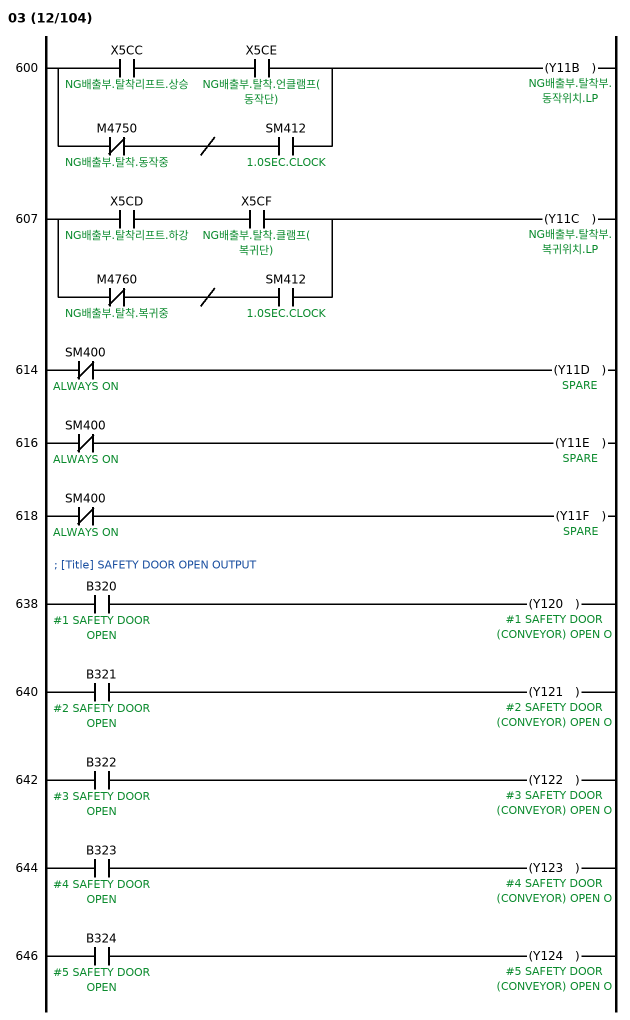
600   LD      X5CC  ; NG배출부.탈착리프트.상승
      AND     X5CE  ; NG배출부.탈착.언클램프(동작단)
      LDI     M4750  ; NG배출부.탈착.동작중
      INV
      AND     SM412  ; 1.0SEC.CLOCK
      ORB
      OUT     Y11B  ; NG배출부.탈착부.동작위치.LP
607   LD      X5CD  ; NG배출부.탈착리프트.하강
      AND     X5CF  ; NG배출부.탈착.클램프(복귀단)
      LDI     M4760  ; NG배출부.탈착.복귀중
      INV
      AND     SM412  ; 1.0SEC.CLOCK
      ORB
      OUT     Y11C  ; NG배출부.탈착부.복귀위치.LP
614   LDI     SM400  ; ALWAYS ON
      OUT     Y11D  ; SPARE
616   LDI     SM400  ; ALWAYS ON
      OUT     Y11E  ; SPARE
618   LDI     SM400  ; ALWAYS ON
      OUT     Y11F  ; SPARE
; [Title] SAFETY DOOR OPEN OUTPUT
638   LD      B320  ; #1 SAFETY DOOR  OPEN
      OUT     Y120  ; #1 SAFETY DOOR (CONVEYOR) OPEN O
640   LD      B321  ; #2 SAFETY DOOR  OPEN
      OUT     Y121  ; #2 SAFETY DOOR (CONVEYOR) OPEN O
642   LD      B322  ; #3 SAFETY DOOR  OPEN
      OUT     Y122  ; #3 SAFETY DOOR (CONVEYOR) OPEN O
644   LD      B323  ; #4 SAFETY DOOR  OPEN
      OUT     Y123  ; #4 SAFETY DOOR (CONVEYOR) OPEN O
646   LD      B324  ; #5 SAFETY DOOR  OPEN
      OUT     Y124  ; #5 SAFETY DOOR (CONVEYOR) OPEN O
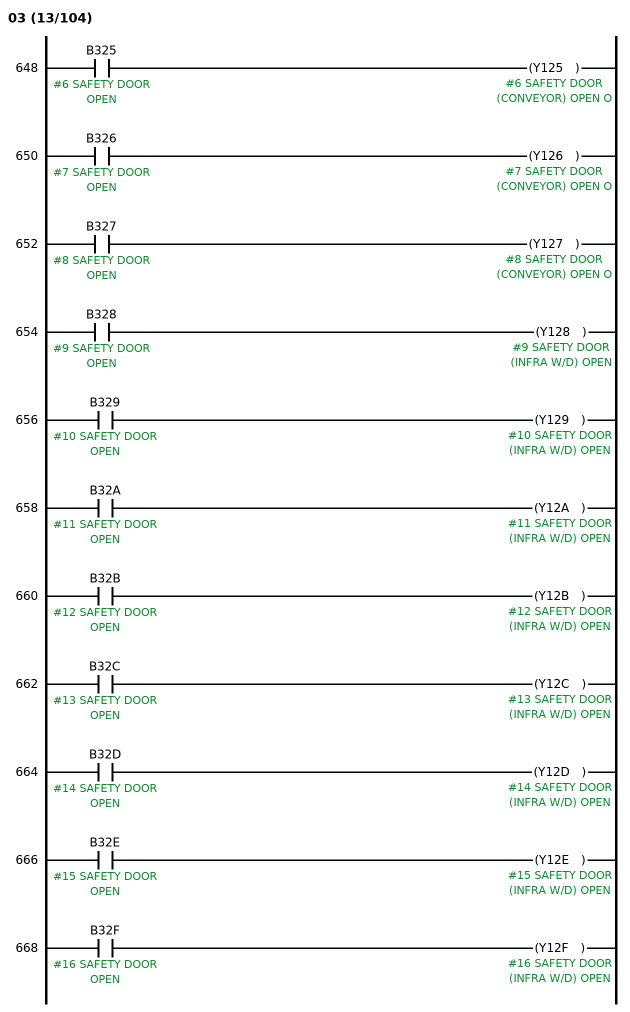
648   LD      B325  ; #6 SAFETY DOOR  OPEN
      OUT     Y125  ; #6 SAFETY DOOR (CONVEYOR) OPEN O
650   LD      B326  ; #7 SAFETY DOOR  OPEN
      OUT     Y126  ; #7 SAFETY DOOR (CONVEYOR) OPEN O
652   LD      B327  ; #8 SAFETY DOOR  OPEN
      OUT     Y127  ; #8 SAFETY DOOR (CONVEYOR) OPEN O
654   LD      B328  ; #9 SAFETY DOOR  OPEN
      OUT     Y128  ; #9 SAFETY DOOR (INFRA W/D) OPEN
656   LD      B329  ; #10 SAFETY DOOR OPEN
      OUT     Y129  ; #10 SAFETY DOOR (INFRA W/D) OPEN
658   LD      B32A  ; #11 SAFETY DOOR OPEN
      OUT     Y12A  ; #11 SAFETY DOOR (INFRA W/D) OPEN
660   LD      B32B  ; #12 SAFETY DOOR OPEN
      OUT     Y12B  ; #12 SAFETY DOOR (INFRA W/D) OPEN
662   LD      B32C  ; #13 SAFETY DOOR OPEN
      OUT     Y12C  ; #13 SAFETY DOOR (INFRA W/D) OPEN
664   LD      B32D  ; #14 SAFETY DOOR OPEN
      OUT     Y12D  ; #14 SAFETY DOOR (INFRA W/D) OPEN
666   LD      B32E  ; #15 SAFETY DOOR OPEN
      OUT     Y12E  ; #15 SAFETY DOOR (INFRA W/D) OPEN
668   LD      B32F  ; #16 SAFETY DOOR OPEN
      OUT     Y12F  ; #16 SAFETY DOOR (INFRA W/D) OPEN
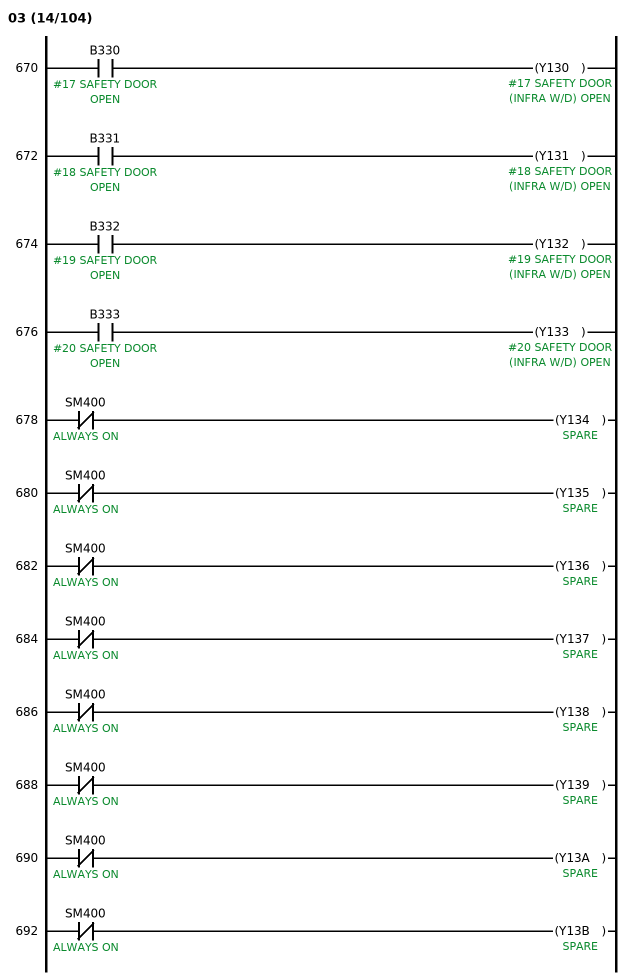
670   LD      B330  ; #17 SAFETY DOOR OPEN
      OUT     Y130  ; #17 SAFETY DOOR (INFRA W/D) OPEN
672   LD      B331  ; #18 SAFETY DOOR OPEN
      OUT     Y131  ; #18 SAFETY DOOR (INFRA W/D) OPEN
674   LD      B332  ; #19 SAFETY DOOR OPEN
      OUT     Y132  ; #19 SAFETY DOOR (INFRA W/D) OPEN
676   LD      B333  ; #20 SAFETY DOOR OPEN
      OUT     Y133  ; #20 SAFETY DOOR (INFRA W/D) OPEN
678   LDI     SM400  ; ALWAYS ON
      OUT     Y134  ; SPARE
680   LDI     SM400  ; ALWAYS ON
      OUT     Y135  ; SPARE
682   LDI     SM400  ; ALWAYS ON
      OUT     Y136  ; SPARE
684   LDI     SM400  ; ALWAYS ON
      OUT     Y137  ; SPARE
686   LDI     SM400  ; ALWAYS ON
      OUT     Y138  ; SPARE
688   LDI     SM400  ; ALWAYS ON
      OUT     Y139  ; SPARE
690   LDI     SM400  ; ALWAYS ON
      OUT     Y13A  ; SPARE
692   LDI     SM400  ; ALWAYS ON
      OUT     Y13B  ; SPARE
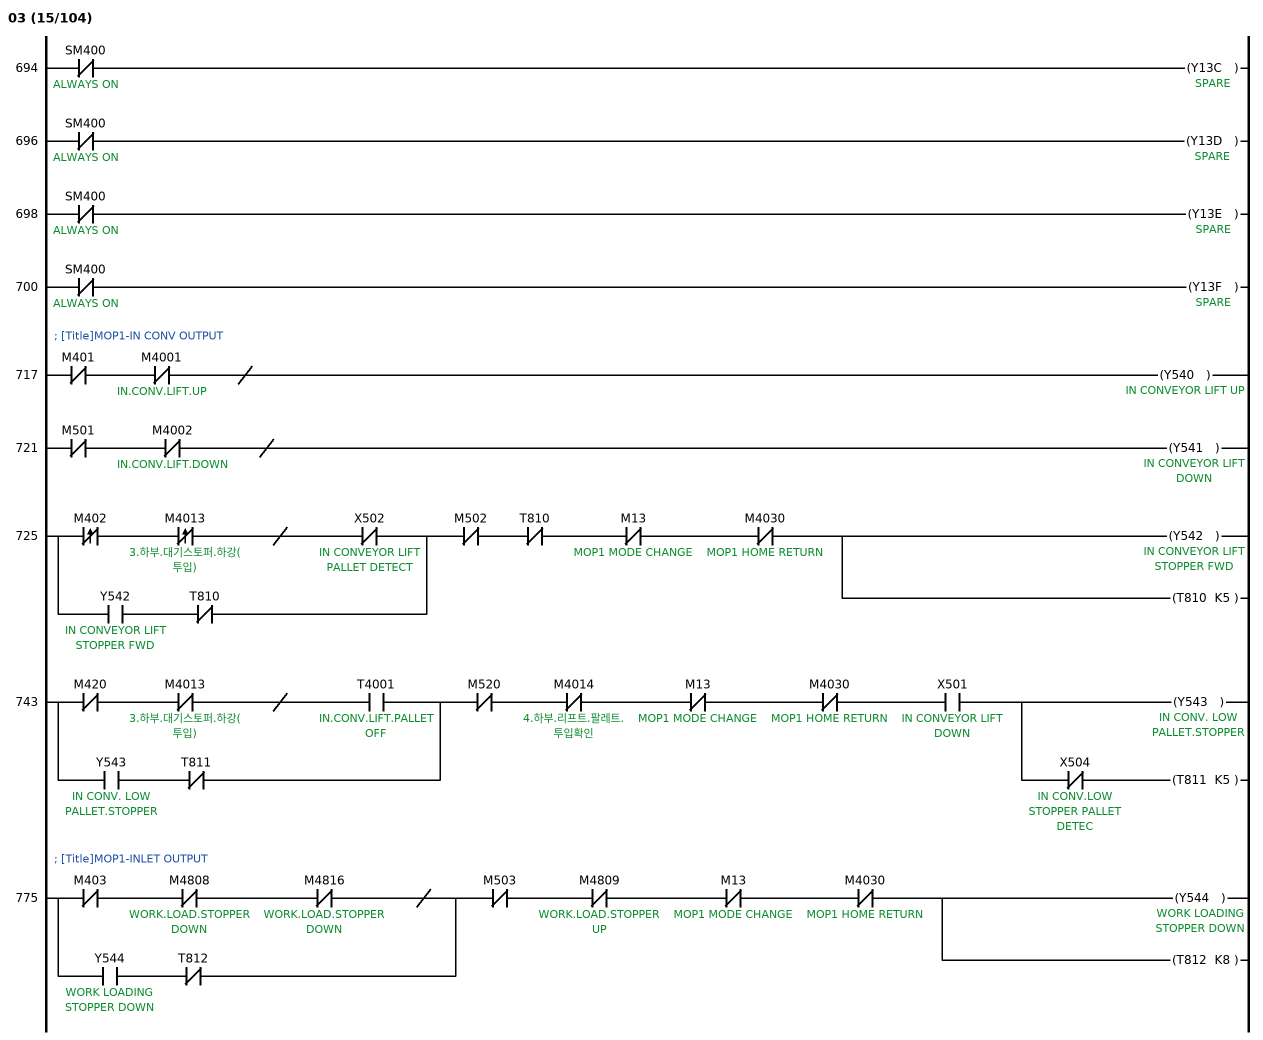
694   LDI     SM400  ; ALWAYS ON
      OUT     Y13C  ; SPARE
696   LDI     SM400  ; ALWAYS ON
      OUT     Y13D  ; SPARE
698   LDI     SM400  ; ALWAYS ON
      OUT     Y13E  ; SPARE
700   LDI     SM400  ; ALWAYS ON
      OUT     Y13F  ; SPARE
; [Title]MOP1-IN CONV OUTPUT
717   LDI     M401
      ANI     M4001  ; IN.CONV.LIFT.UP
      INV
      OUT     Y540  ; IN CONVEYOR LIFT UP
721   LDI     M501
      ANI     M4002  ; IN.CONV.LIFT.DOWN
      INV
      OUT     Y541  ; IN CONVEYOR LIFT DOWN
725   LDPI    M402
      ANDPI   M4013  ; 3.하부.대기스토퍼.하강(투입)
      INV
      ANI     X502  ; IN CONVEYOR LIFT PALLET DETECT
      LD      Y542  ; IN CONVEYOR LIFT STOPPER FWD
      ANI     T810
      ORB
      ANI     M502
      ANI     T810
      ANI     M13  ; MOP1 MODE CHANGE
      ANI     M4030  ; MOP1 HOME RETURN
      OUT     Y542  ; IN CONVEYOR LIFT STOPPER FWD
      OUT     T810 K5
743   LDI     M420
      ANI     M4013  ; 3.하부.대기스토퍼.하강(투입)
      INV
      AND     T4001  ; IN.CONV.LIFT.PALLET OFF
      LD      Y543  ; IN CONV. LOW PALLET.STOPPER
      ANI     T811
      ORB
      ANI     M520
      ANI     M4014  ; 4.하부.리프트.팔레트.투입확인
      ANI     M13  ; MOP1 MODE CHANGE
      ANI     M4030  ; MOP1 HOME RETURN
      AND     X501  ; IN CONVEYOR LIFT DOWN
      OUT     Y543  ; IN CONV. LOW PALLET.STOPPER
      ANI     X504  ; IN CONV.LOW STOPPER PALLET DETEC
      OUT     T811 K5
; [Title]MOP1-INLET OUTPUT
775   LDI     M403
      ANI     M4808  ; WORK.LOAD.STOPPER DOWN
      ANI     M4816  ; WORK.LOAD.STOPPER DOWN
      INV
      LD      Y544  ; WORK LOADING STOPPER DOWN
      ANI     T812
      ORB
      ANI     M503
      ANI     M4809  ; WORK.LOAD.STOPPER UP
      ANI     M13  ; MOP1 MODE CHANGE
      ANI     M4030  ; MOP1 HOME RETURN
      OUT     Y544  ; WORK LOADING STOPPER DOWN
      OUT     T812 K8
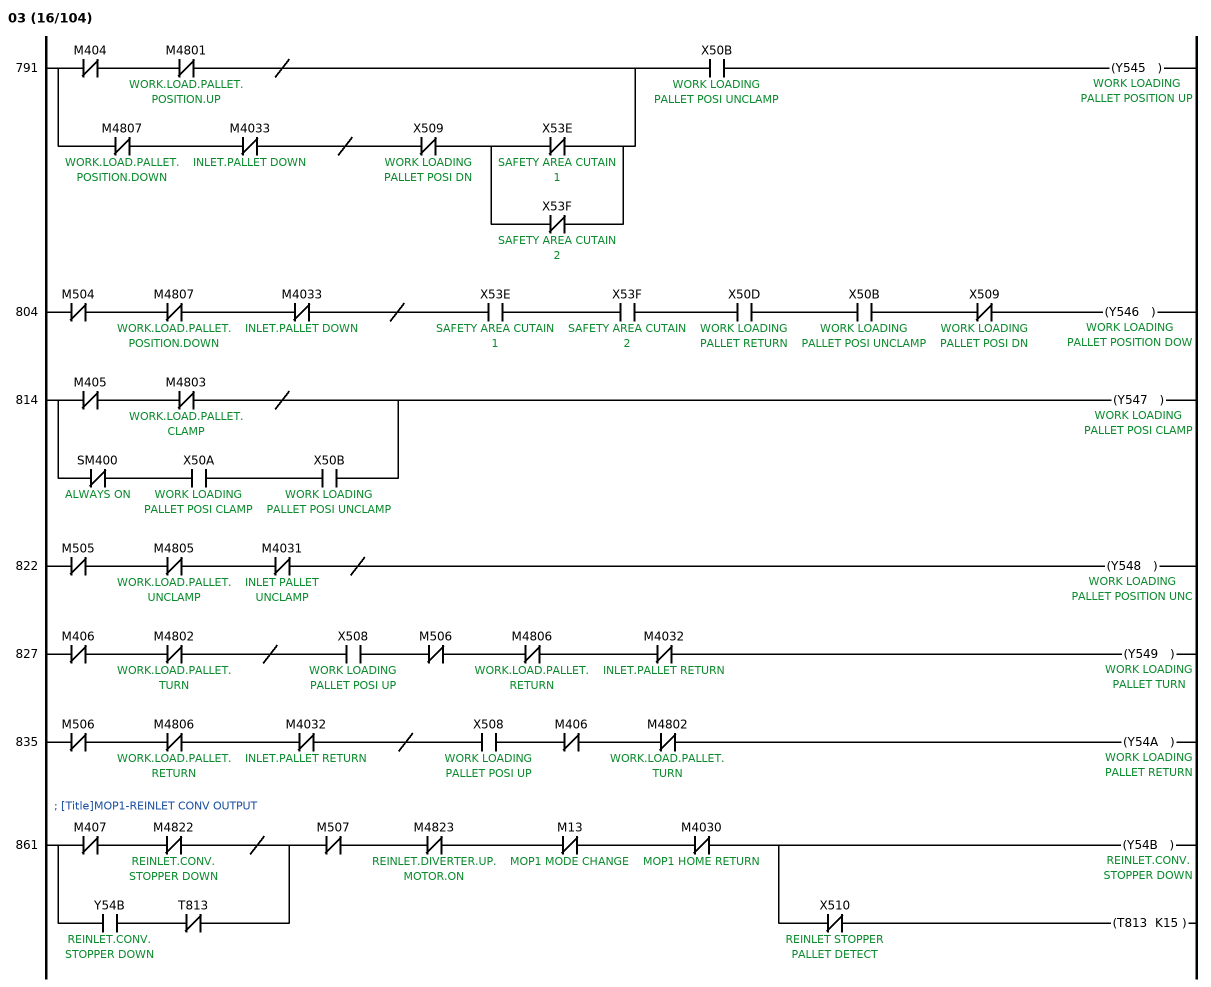
791   LDI     M404
      ANI     M4801  ; WORK.LOAD.PALLET.POSITION.UP
      INV
      LDI     M4807  ; WORK.LOAD.PALLET.POSITION.DOWN
      ANI     M4033  ; INLET.PALLET DOWN
      INV
      ANI     X509  ; WORK LOADING PALLET POSI DN
      LDI     X53E  ; SAFETY AREA CUTAIN 1
      ORI     X53F  ; SAFETY AREA CUTAIN 2
      ANB
      ORB
      AND     X50B  ; WORK LOADING PALLET POSI UNCLAMP
      OUT     Y545  ; WORK LOADING PALLET POSITION UP
804   LDI     M504
      ANI     M4807  ; WORK.LOAD.PALLET.POSITION.DOWN
      ANI     M4033  ; INLET.PALLET DOWN
      INV
      AND     X53E  ; SAFETY AREA CUTAIN 1
      AND     X53F  ; SAFETY AREA CUTAIN 2
      AND     X50D  ; WORK LOADING PALLET RETURN
      AND     X50B  ; WORK LOADING PALLET POSI UNCLAMP
      ANI     X509  ; WORK LOADING PALLET POSI DN
      OUT     Y546  ; WORK LOADING PALLET POSITION DOW
814   LDI     M405
      ANI     M4803  ; WORK.LOAD.PALLET.CLAMP
      INV
      LDI     SM400  ; ALWAYS ON
      AND     X50A  ; WORK LOADING PALLET POSI CLAMP
      AND     X50B  ; WORK LOADING PALLET POSI UNCLAMP
      ORB
      OUT     Y547  ; WORK LOADING PALLET POSI CLAMP
822   LDI     M505
      ANI     M4805  ; WORK.LOAD.PALLET.UNCLAMP
      ANI     M4031  ; INLET PALLET UNCLAMP
      INV
      OUT     Y548  ; WORK LOADING PALLET POSITION UNC
827   LDI     M406
      ANI     M4802  ; WORK.LOAD.PALLET.TURN
      INV
      AND     X508  ; WORK LOADING PALLET POSI UP
      ANI     M506
      ANI     M4806  ; WORK.LOAD.PALLET.RETURN
      ANI     M4032  ; INLET.PALLET RETURN
      OUT     Y549  ; WORK LOADING PALLET TURN
835   LDI     M506
      ANI     M4806  ; WORK.LOAD.PALLET.RETURN
      ANI     M4032  ; INLET.PALLET RETURN
      INV
      AND     X508  ; WORK LOADING PALLET POSI UP
      ANI     M406
      ANI     M4802  ; WORK.LOAD.PALLET.TURN
      OUT     Y54A  ; WORK LOADING PALLET RETURN
; [Title]MOP1-REINLET CONV OUTPUT
861   LDI     M407
      ANI     M4822  ; REINLET.CONV.STOPPER DOWN
      INV
      LD      Y54B  ; REINLET.CONV.STOPPER DOWN
      ANI     T813
      ORB
      ANI     M507
      ANI     M4823  ; REINLET.DIVERTER.UP.MOTOR.ON
      ANI     M13  ; MOP1 MODE CHANGE
      ANI     M4030  ; MOP1 HOME RETURN
      OUT     Y54B  ; REINLET.CONV.STOPPER DOWN
      ANI     X510  ; REINLET STOPPER PALLET DETECT
      OUT     T813 K15
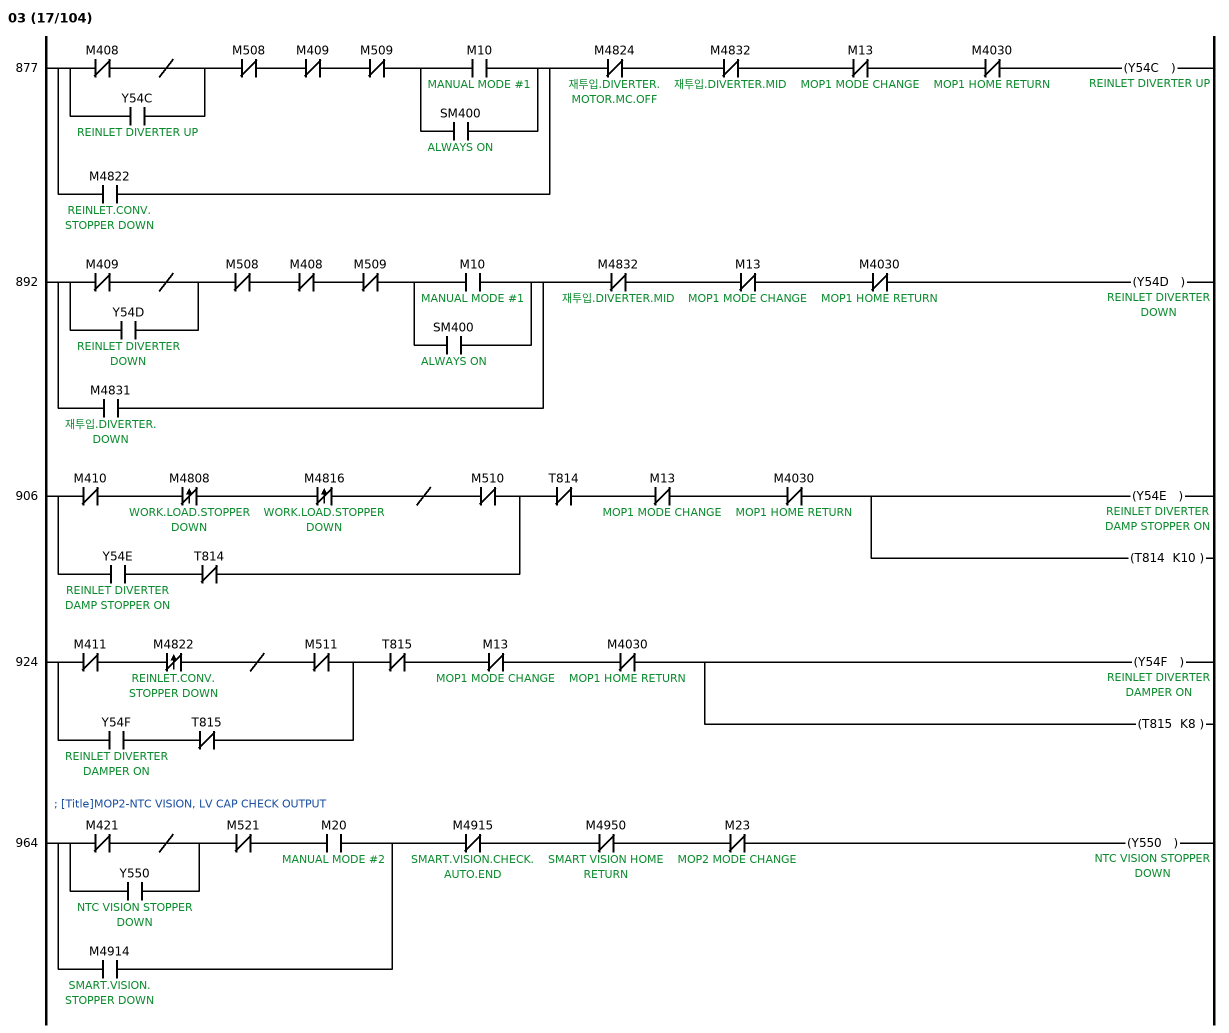
877   LDI     M408
      INV
      OR      Y54C  ; REINLET DIVERTER UP
      ANI     M508
      ANI     M409
      ANI     M509
      LD      M10  ; MANUAL MODE #1
      OR      SM400  ; ALWAYS ON
      ANB
      OR      M4822  ; REINLET.CONV.STOPPER DOWN
      ANI     M4824  ; 재투입.DIVERTER.MOTOR.MC.OFF
      ANI     M4832  ; 재투입.DIVERTER.MID
      ANI     M13  ; MOP1 MODE CHANGE
      ANI     M4030  ; MOP1 HOME RETURN
      OUT     Y54C  ; REINLET DIVERTER UP
892   LDI     M409
      INV
      OR      Y54D  ; REINLET DIVERTER DOWN
      ANI     M508
      ANI     M408
      ANI     M509
      LD      M10  ; MANUAL MODE #1
      OR      SM400  ; ALWAYS ON
      ANB
      OR      M4831  ; 재투입.DIVERTER.DOWN
      ANI     M4832  ; 재투입.DIVERTER.MID
      ANI     M13  ; MOP1 MODE CHANGE
      ANI     M4030  ; MOP1 HOME RETURN
      OUT     Y54D  ; REINLET DIVERTER DOWN
906   LDI     M410
      ANDPI   M4808  ; WORK.LOAD.STOPPER DOWN
      ANDPI   M4816  ; WORK.LOAD.STOPPER DOWN
      INV
      ANI     M510
      LD      Y54E  ; REINLET DIVERTER DAMP STOPPER ON
      ANI     T814
      ORB
      ANI     T814
      ANI     M13  ; MOP1 MODE CHANGE
      ANI     M4030  ; MOP1 HOME RETURN
      OUT     Y54E  ; REINLET DIVERTER DAMP STOPPER ON
      OUT     T814 K10
924   LDI     M411
      ANDPI   M4822  ; REINLET.CONV.STOPPER DOWN
      INV
      ANI     M511
      LD      Y54F  ; REINLET DIVERTER DAMPER ON
      ANI     T815
      ORB
      ANI     T815
      ANI     M13  ; MOP1 MODE CHANGE
      ANI     M4030  ; MOP1 HOME RETURN
      OUT     Y54F  ; REINLET DIVERTER DAMPER ON
      OUT     T815 K8
; [Title]MOP2-NTC VISION, LV CAP CHECK OUTPUT
964   LDI     M421
      INV
      OR      Y550  ; NTC VISION STOPPER DOWN
      ANI     M521
      AND     M20  ; MANUAL MODE #2
      OR      M4914  ; SMART.VISION.STOPPER DOWN
      ANI     M4915  ; SMART.VISION.CHECK.AUTO.END
      ANI     M4950  ; SMART VISION HOME RETURN
      ANI     M23  ; MOP2 MODE CHANGE
      OUT     Y550  ; NTC VISION STOPPER DOWN
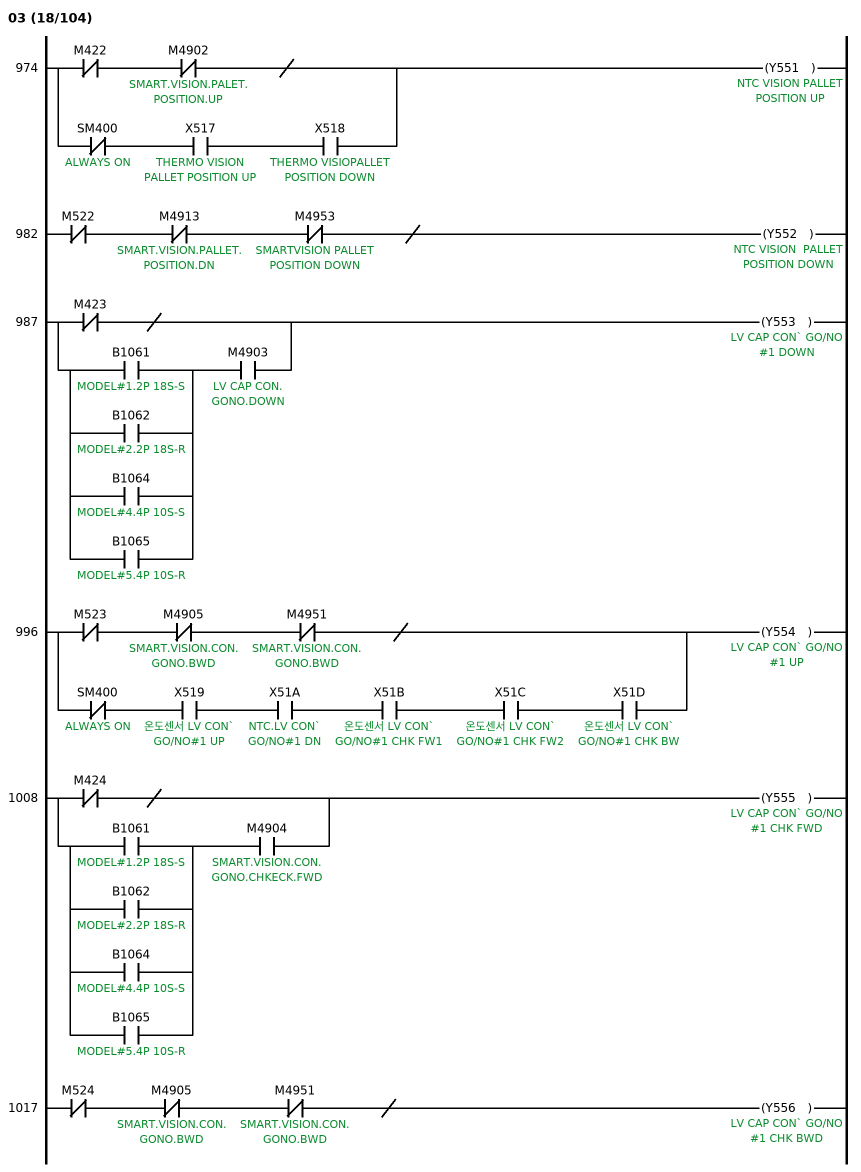
974   LDI     M422
      ANI     M4902  ; SMART.VISION.PALET.POSITION.UP
      INV
      LDI     SM400  ; ALWAYS ON
      AND     X517  ; THERMO VISION PALLET POSITION UP
      AND     X518  ; THERMO VISIOPALLET POSITION DOWN
      ORB
      OUT     Y551  ; NTC VISION PALLET POSITION UP
982   LDI     M522
      ANI     M4913  ; SMART.VISION.PALLET.POSITION.DN
      ANI     M4953  ; SMARTVISION PALLET POSITION DOWN
      INV
      OUT     Y552  ; NTC VISION  PALLET POSITION DOWN
987   LDI     M423
      INV
      LD      B1061  ; MODEL#1.2P 18S-S
      OR      B1062  ; MODEL#2.2P 18S-R
      OR      B1064  ; MODEL#4.4P 10S-S
      OR      B1065  ; MODEL#5.4P 10S-R
      AND     M4903  ; LV CAP CON. GONO.DOWN
      ORB
      OUT     Y553  ; LV CAP CON` GO/NO #1 DOWN
996   LDI     M523
      ANI     M4905  ; SMART.VISION.CON.GONO.BWD
      ANI     M4951  ; SMART.VISION.CON.GONO.BWD
      INV
      LDI     SM400  ; ALWAYS ON
      AND     X519  ; 온도센서 LV CON` GO/NO#1 UP
      AND     X51A  ; NTC.LV CON` GO/NO#1 DN
      AND     X51B  ; 온도센서 LV CON` GO/NO#1 CHK FW1
      AND     X51C  ; 온도센서 LV CON` GO/NO#1 CHK FW2
      AND     X51D  ; 온도센서 LV CON` GO/NO#1 CHK BW
      ORB
      OUT     Y554  ; LV CAP CON` GO/NO #1 UP
1008  LDI     M424
      INV
      LD      B1061  ; MODEL#1.2P 18S-S
      OR      B1062  ; MODEL#2.2P 18S-R
      OR      B1064  ; MODEL#4.4P 10S-S
      OR      B1065  ; MODEL#5.4P 10S-R
      AND     M4904  ; SMART.VISION.CON.GONO.CHKECK.FWD
      ORB
      OUT     Y555  ; LV CAP CON` GO/NO #1 CHK FWD
1017  LDI     M524
      ANI     M4905  ; SMART.VISION.CON.GONO.BWD
      ANI     M4951  ; SMART.VISION.CON.GONO.BWD
      INV
      OUT     Y556  ; LV CAP CON` GO/NO #1 CHK BWD
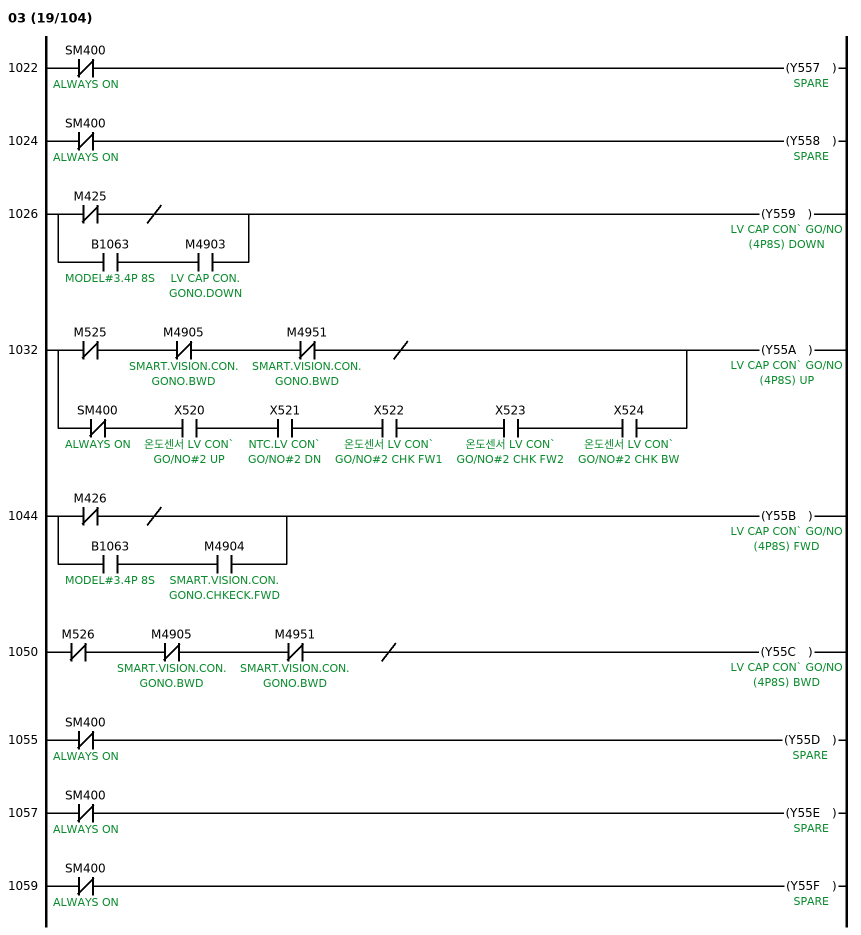
1022  LDI     SM400  ; ALWAYS ON
      OUT     Y557  ; SPARE
1024  LDI     SM400  ; ALWAYS ON
      OUT     Y558  ; SPARE
1026  LDI     M425
      INV
      LD      B1063  ; MODEL#3.4P 8S
      AND     M4903  ; LV CAP CON. GONO.DOWN
      ORB
      OUT     Y559  ; LV CAP CON` GO/NO (4P8S) DOWN
1032  LDI     M525
      ANI     M4905  ; SMART.VISION.CON.GONO.BWD
      ANI     M4951  ; SMART.VISION.CON.GONO.BWD
      INV
      LDI     SM400  ; ALWAYS ON
      AND     X520  ; 온도센서 LV CON` GO/NO#2 UP
      AND     X521  ; NTC.LV CON` GO/NO#2 DN
      AND     X522  ; 온도센서 LV CON` GO/NO#2 CHK FW1
      AND     X523  ; 온도센서 LV CON` GO/NO#2 CHK FW2
      AND     X524  ; 온도센서 LV CON` GO/NO#2 CHK BW
      ORB
      OUT     Y55A  ; LV CAP CON` GO/NO (4P8S) UP
1044  LDI     M426
      INV
      LD      B1063  ; MODEL#3.4P 8S
      AND     M4904  ; SMART.VISION.CON.GONO.CHKECK.FWD
      ORB
      OUT     Y55B  ; LV CAP CON` GO/NO (4P8S) FWD
1050  LDI     M526
      ANI     M4905  ; SMART.VISION.CON.GONO.BWD
      ANI     M4951  ; SMART.VISION.CON.GONO.BWD
      INV
      OUT     Y55C  ; LV CAP CON` GO/NO (4P8S) BWD
1055  LDI     SM400  ; ALWAYS ON
      OUT     Y55D  ; SPARE
1057  LDI     SM400  ; ALWAYS ON
      OUT     Y55E  ; SPARE
1059  LDI     SM400  ; ALWAYS ON
      OUT     Y55F  ; SPARE
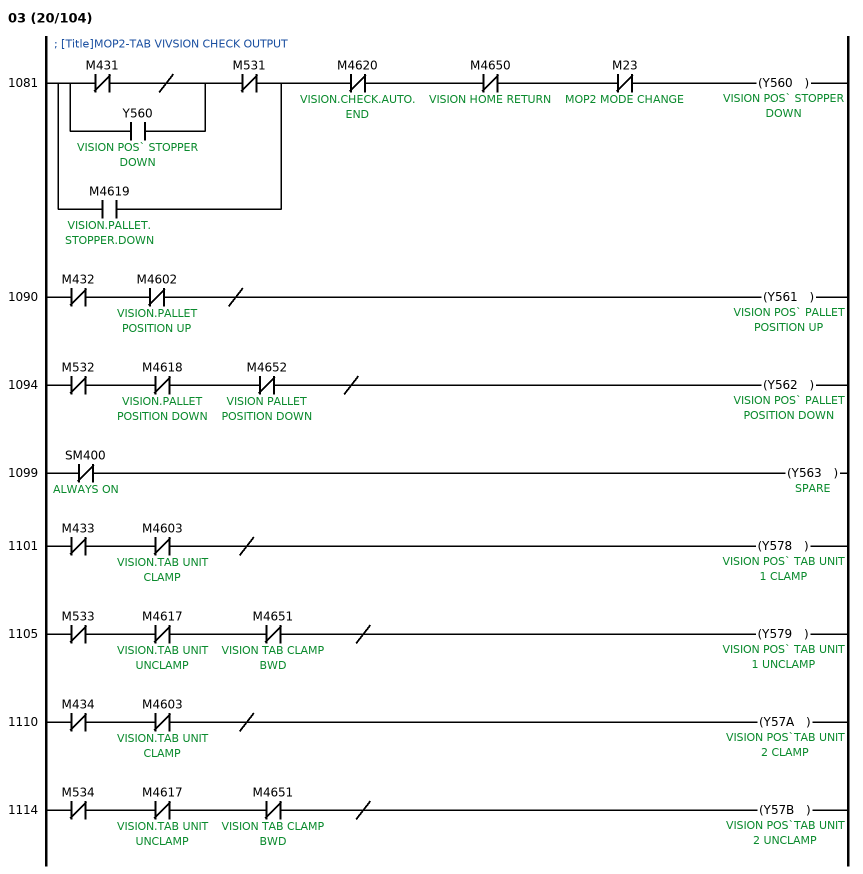
; [Title]MOP2-TAB VIVSION CHECK OUTPUT
1081  LDI     M431
      INV
      OR      Y560  ; VISION POS` STOPPER DOWN
      ANI     M531
      OR      M4619  ; VISION.PALLET.STOPPER.DOWN
      ANI     M4620  ; VISION.CHECK.AUTO.END
      ANI     M4650  ; VISION HOME RETURN
      ANI     M23  ; MOP2 MODE CHANGE
      OUT     Y560  ; VISION POS` STOPPER DOWN
1090  LDI     M432
      ANI     M4602  ; VISION.PALLET POSITION UP
      INV
      OUT     Y561  ; VISION POS` PALLET POSITION UP
1094  LDI     M532
      ANI     M4618  ; VISION.PALLET POSITION DOWN
      ANI     M4652  ; VISION PALLET POSITION DOWN
      INV
      OUT     Y562  ; VISION POS` PALLET POSITION DOWN
1099  LDI     SM400  ; ALWAYS ON
      OUT     Y563  ; SPARE
1101  LDI     M433
      ANI     M4603  ; VISION.TAB UNIT CLAMP
      INV
      OUT     Y578  ; VISION POS` TAB UNIT 1 CLAMP
1105  LDI     M533
      ANI     M4617  ; VISION.TAB UNIT UNCLAMP
      ANI     M4651  ; VISION TAB CLAMP BWD
      INV
      OUT     Y579  ; VISION POS` TAB UNIT 1 UNCLAMP
1110  LDI     M434
      ANI     M4603  ; VISION.TAB UNIT CLAMP
      INV
      OUT     Y57A  ; VISION POS`TAB UNIT 2 CLAMP
1114  LDI     M534
      ANI     M4617  ; VISION.TAB UNIT UNCLAMP
      ANI     M4651  ; VISION TAB CLAMP BWD
      INV
      OUT     Y57B  ; VISION POS`TAB UNIT 2 UNCLAMP
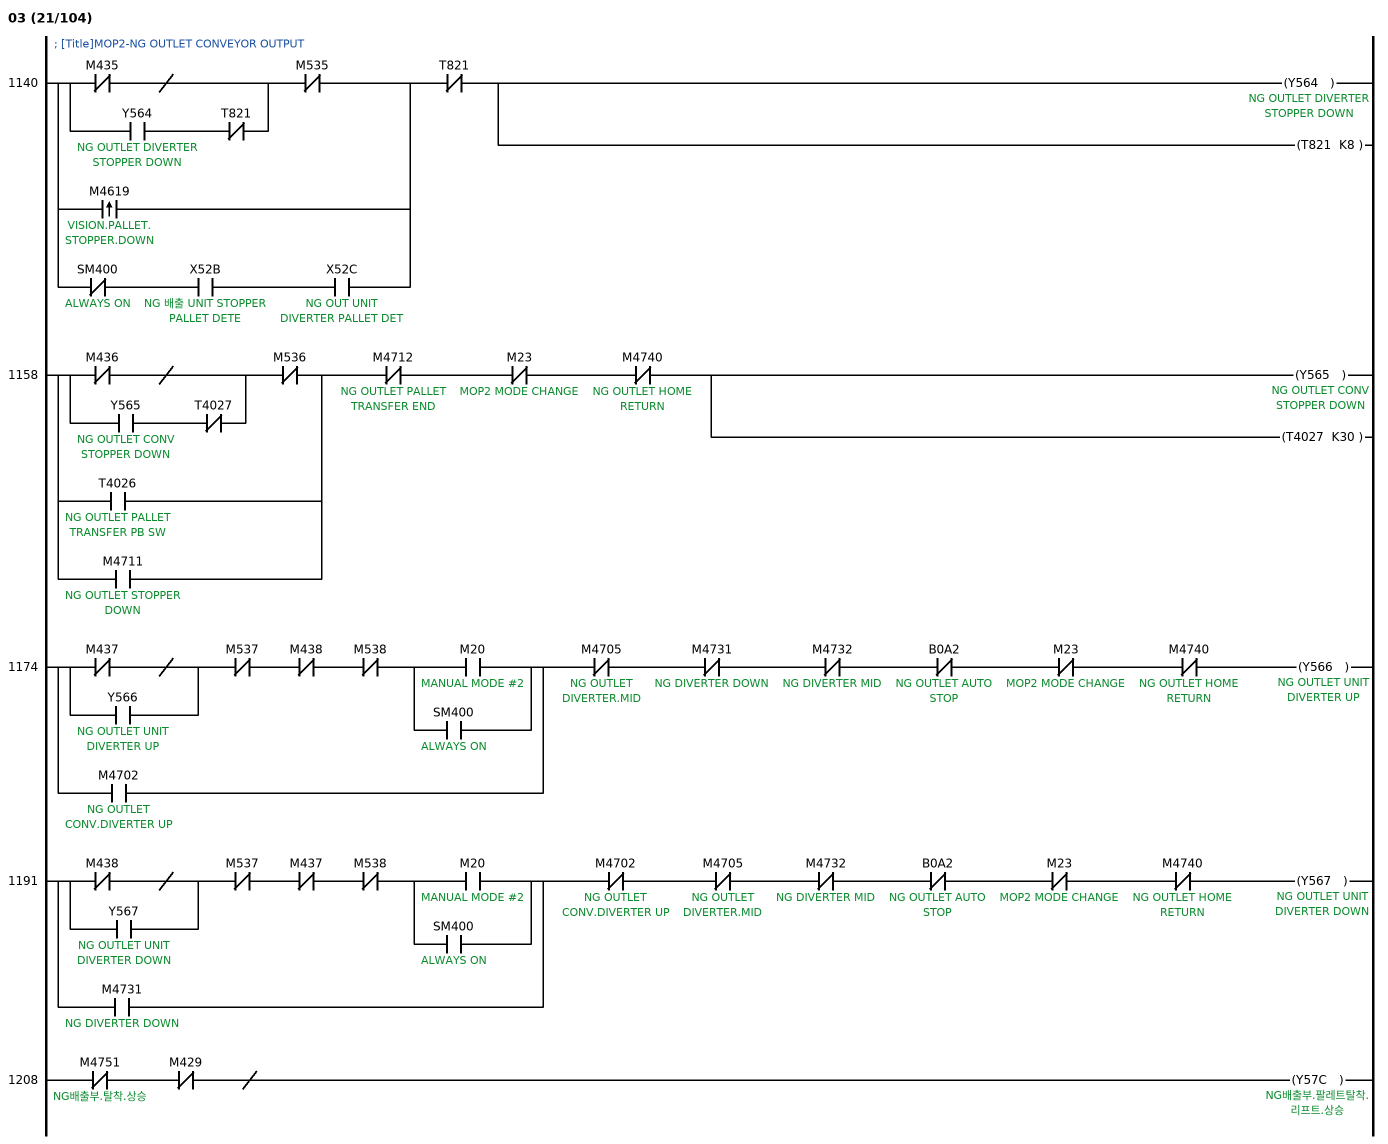
; [Title]MOP2-NG OUTLET CONVEYOR OUTPUT
1140  LDI     M435
      INV
      LD      Y564  ; NG OUTLET DIVERTER STOPPER DOWN
      ANI     T821
      ORB
      ANI     M535
      ORP     M4619  ; VISION.PALLET.STOPPER.DOWN
      LDI     SM400  ; ALWAYS ON
      AND     X52B  ; NG 배출 UNIT STOPPER PALLET DETE
      AND     X52C  ; NG OUT UNIT DIVERTER PALLET DET
      ORB
      ANI     T821
      OUT     Y564  ; NG OUTLET DIVERTER STOPPER DOWN
      OUT     T821 K8
1158  LDI     M436
      INV
      LD      Y565  ; NG OUTLET CONV STOPPER DOWN
      ANI     T4027
      ORB
      ANI     M536
      OR      T4026  ; NG OUTLET PALLET TRANSFER PB SW
      OR      M4711  ; NG OUTLET STOPPER DOWN
      ANI     M4712  ; NG OUTLET PALLET TRANSFER END
      ANI     M23  ; MOP2 MODE CHANGE
      ANI     M4740  ; NG OUTLET HOME RETURN
      OUT     Y565  ; NG OUTLET CONV STOPPER DOWN
      OUT     T4027 K30
1174  LDI     M437
      INV
      OR      Y566  ; NG OUTLET UNIT DIVERTER UP
      ANI     M537
      ANI     M438
      ANI     M538
      LD      M20  ; MANUAL MODE #2
      OR      SM400  ; ALWAYS ON
      ANB
      OR      M4702  ; NG OUTLET CONV.DIVERTER UP
      ANI     M4705  ; NG OUTLET DIVERTER.MID
      ANI     M4731  ; NG DIVERTER DOWN
      ANI     M4732  ; NG DIVERTER MID
      ANI     B0A2  ; NG OUTLET AUTO STOP
      ANI     M23  ; MOP2 MODE CHANGE
      ANI     M4740  ; NG OUTLET HOME RETURN
      OUT     Y566  ; NG OUTLET UNIT DIVERTER UP
1191  LDI     M438
      INV
      OR      Y567  ; NG OUTLET UNIT DIVERTER DOWN
      ANI     M537
      ANI     M437
      ANI     M538
      LD      M20  ; MANUAL MODE #2
      OR      SM400  ; ALWAYS ON
      ANB
      OR      M4731  ; NG DIVERTER DOWN
      ANI     M4702  ; NG OUTLET CONV.DIVERTER UP
      ANI     M4705  ; NG OUTLET DIVERTER.MID
      ANI     M4732  ; NG DIVERTER MID
      ANI     B0A2  ; NG OUTLET AUTO STOP
      ANI     M23  ; MOP2 MODE CHANGE
      ANI     M4740  ; NG OUTLET HOME RETURN
      OUT     Y567  ; NG OUTLET UNIT DIVERTER DOWN
1208  LDI     M4751  ; NG배출부.탈착.상승
      ANI     M429
      INV
      OUT     Y57C  ; NG배출부.팔레트탈착.리프트.상승
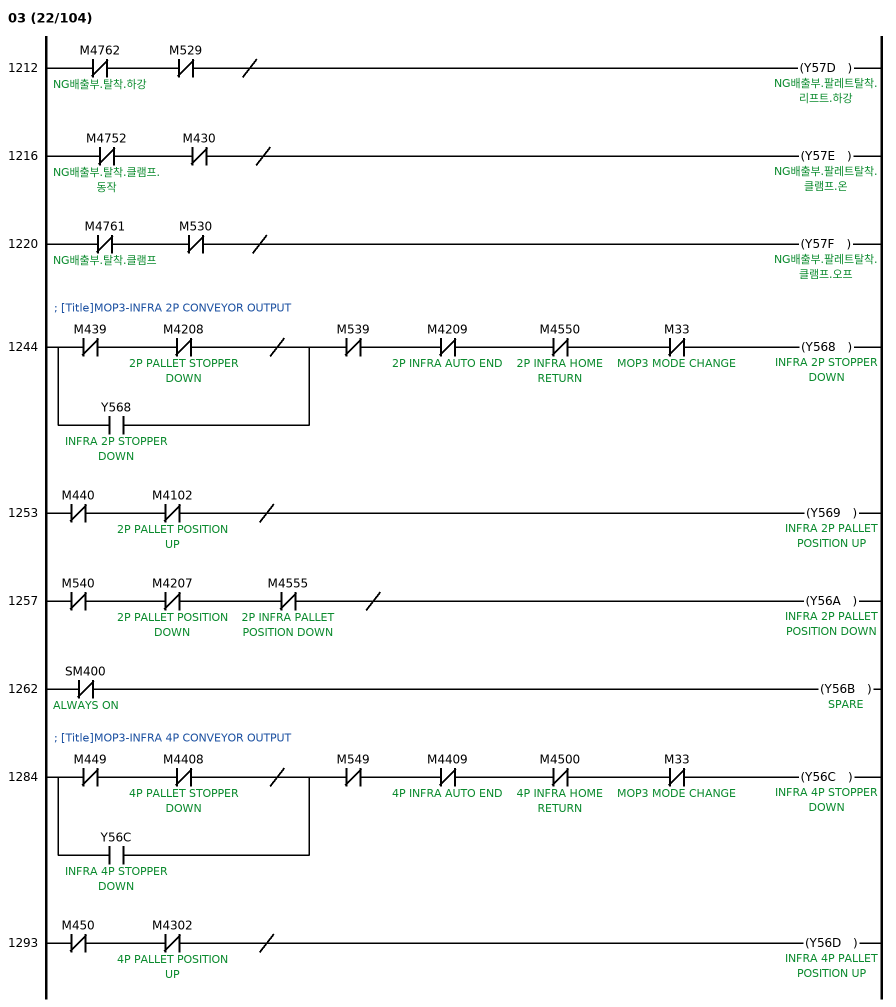
1212  LDI     M4762  ; NG배출부.탈착.하강
      ANI     M529
      INV
      OUT     Y57D  ; NG배출부.팔레트탈착.리프트.하강
1216  LDI     M4752  ; NG배출부.탈착.클램프.동작
      ANI     M430
      INV
      OUT     Y57E  ; NG배출부.팔레트탈착.클램프.온
1220  LDI     M4761  ; NG배출부.탈착.클램프
      ANI     M530
      INV
      OUT     Y57F  ; NG배출부.팔레트탈착.클램프.오프
; [Title]MOP3-INFRA 2P CONVEYOR OUTPUT
1244  LDI     M439
      ANI     M4208  ; 2P PALLET STOPPER DOWN
      INV
      OR      Y568  ; INFRA 2P STOPPER DOWN
      ANI     M539
      ANI     M4209  ; 2P INFRA AUTO END
      ANI     M4550  ; 2P INFRA HOME RETURN
      ANI     M33  ; MOP3 MODE CHANGE
      OUT     Y568  ; INFRA 2P STOPPER DOWN
1253  LDI     M440
      ANI     M4102  ; 2P PALLET POSITION UP
      INV
      OUT     Y569  ; INFRA 2P PALLET POSITION UP
1257  LDI     M540
      ANI     M4207  ; 2P PALLET POSITION DOWN
      ANI     M4555  ; 2P INFRA PALLET POSITION DOWN
      INV
      OUT     Y56A  ; INFRA 2P PALLET POSITION DOWN
1262  LDI     SM400  ; ALWAYS ON
      OUT     Y56B  ; SPARE
; [Title]MOP3-INFRA 4P CONVEYOR OUTPUT
1284  LDI     M449
      ANI     M4408  ; 4P PALLET STOPPER DOWN
      INV
      OR      Y56C  ; INFRA 4P STOPPER DOWN
      ANI     M549
      ANI     M4409  ; 4P INFRA AUTO END
      ANI     M4500  ; 4P INFRA HOME RETURN
      ANI     M33  ; MOP3 MODE CHANGE
      OUT     Y56C  ; INFRA 4P STOPPER DOWN
1293  LDI     M450
      ANI     M4302  ; 4P PALLET POSITION UP
      INV
      OUT     Y56D  ; INFRA 4P PALLET POSITION UP
